; END LAYER 35
LIN {X -34.33, Y -49.21, Z 72.0, A 0, B 90, C 0} C_DIS
WAIT SEC 3
LIN {X -34.33, Y -49.21, Z 74.0, A 0, B 90, C 0} C_DIS
$OUT[1] = TRUE
WAIT SEC 0.8
LIN {X -34.33, Y -49.21, Z 74.0, A 0, B 90, C 0} C_DIS
LIN {X -34.33, Y -49.21, Z 74.0, A 0, B 90, C 0} C_DIS
LIN {X -32.91, Y -50.13, Z 74.0, A 0, B 90, C 0} C_DIS
LIN {X -31.1, Y -51.31, Z 74.0, A 0, B 90, C 0} C_DIS
LIN {X -29.63, Y -52.14, Z 74.0, A 0, B 90, C 0} C_DIS
LIN {X -27.75, Y -53.2, Z 74.0, A 0, B 90, C 0} C_DIS
LIN {X -26.23, Y -53.93, Z 74.0, A 0, B 90, C 0} C_DIS
LIN {X -24.29, Y -54.86, Z 74.0, A 0, B 90, C 0} C_DIS
LIN {X -22.72, Y -55.5, Z 74.0, A 0, B 90, C 0} C_DIS
LIN {X -20.72, Y -56.31, Z 74.0, A 0, B 90, C 0} C_DIS
LIN {X -19.12, Y -56.84, Z 74.0, A 0, B 90, C 0} C_DIS
LIN {X -17.07, Y -57.52, Z 74.0, A 0, B 90, C 0} C_DIS
LIN {X -15.43, Y -57.95, Z 74.0, A 0, B 90, C 0} C_DIS
LIN {X -13.35, Y -58.5, Z 74.0, A 0, B 90, C 0} C_DIS
LIN {X -11.69, Y -58.82, Z 74.0, A 0, B 90, C 0} C_DIS
LIN {X -9.58, Y -59.23, Z 74.0, A 0, B 90, C 0} C_DIS
LIN {X -7.9, Y -59.45, Z 74.0, A 0, B 90, C 0} C_DIS
LIN {X -5.76, Y -59.72, Z 74.0, A 0, B 90, C 0} C_DIS
LIN {X -4.07, Y -59.83, Z 74.0, A 0, B 90, C 0} C_DIS
LIN {X -1.92, Y -59.97, Z 74.0, A 0, B 90, C 0} C_DIS
LIN {X -0.23, Y -59.97, Z 74.0, A 0, B 90, C 0} C_DIS
LIN {X 1.92, Y -59.97, Z 74.0, A 0, B 90, C 0} C_DIS
LIN {X 3.61, Y -59.86, Z 74.0, A 0, B 90, C 0} C_DIS
LIN {X 5.76, Y -59.72, Z 74.0, A 0, B 90, C 0} C_DIS
LIN {X 7.44, Y -59.51, Z 74.0, A 0, B 90, C 0} C_DIS
LIN {X 9.58, Y -59.23, Z 74.0, A 0, B 90, C 0} C_DIS
LIN {X 11.24, Y -58.91, Z 74.0, A 0, B 90, C 0} C_DIS
LIN {X 13.35, Y -58.5, Z 74.0, A 0, B 90, C 0} C_DIS
LIN {X 14.99, Y -58.07, Z 74.0, A 0, B 90, C 0} C_DIS
LIN {X 17.07, Y -57.52, Z 74.0, A 0, B 90, C 0} C_DIS
LIN {X 18.68, Y -56.99, Z 74.0, A 0, B 90, C 0} C_DIS
LIN {X 20.72, Y -56.31, Z 74.0, A 0, B 90, C 0} C_DIS
LIN {X 22.29, Y -55.67, Z 74.0, A 0, B 90, C 0} C_DIS
LIN {X 24.29, Y -54.86, Z 74.0, A 0, B 90, C 0} C_DIS
LIN {X 25.81, Y -54.13, Z 74.0, A 0, B 90, C 0} C_DIS
LIN {X 27.75, Y -53.2, Z 74.0, A 0, B 90, C 0} C_DIS
LIN {X 29.23, Y -52.37, Z 74.0, A 0, B 90, C 0} C_DIS
LIN {X 31.1, Y -51.31, Z 74.0, A 0, B 90, C 0} C_DIS
LIN {X 32.52, Y -50.39, Z 74.0, A 0, B 90, C 0} C_DIS
LIN {X 34.33, Y -49.21, Z 74.0, A 0, B 90, C 0} C_DIS
LIN {X 35.68, Y -48.2, Z 74.0, A 0, B 90, C 0} C_DIS
LIN {X 37.41, Y -46.91, Z 74.0, A 0, B 90, C 0} C_DIS
LIN {X 38.7, Y -45.81, Z 74.0, A 0, B 90, C 0} C_DIS
LIN {X 40.34, Y -44.42, Z 74.0, A 0, B 90, C 0} C_DIS
LIN {X 41.55, Y -43.24, Z 74.0, A 0, B 90, C 0} C_DIS
LIN {X 43.1, Y -41.74, Z 74.0, A 0, B 90, C 0} C_DIS
LIN {X 44.24, Y -40.49, Z 74.0, A 0, B 90, C 0} C_DIS
LIN {X 45.69, Y -38.89, Z 74.0, A 0, B 90, C 0} C_DIS
LIN {X 46.74, Y -37.57, Z 74.0, A 0, B 90, C 0} C_DIS
LIN {X 48.08, Y -35.89, Z 74.0, A 0, B 90, C 0} C_DIS
LIN {X 49.05, Y -34.5, Z 74.0, A 0, B 90, C 0} C_DIS
LIN {X 50.29, Y -32.73, Z 74.0, A 0, B 90, C 0} C_DIS
LIN {X 51.16, Y -31.28, Z 74.0, A 0, B 90, C 0} C_DIS
LIN {X 52.28, Y -29.44, Z 74.0, A 0, B 90, C 0} C_DIS
LIN {X 53.06, Y -27.94, Z 74.0, A 0, B 90, C 0} C_DIS
LIN {X 54.06, Y -26.03, Z 74.0, A 0, B 90, C 0} C_DIS
LIN {X 54.74, Y -24.49, Z 74.0, A 0, B 90, C 0} C_DIS
LIN {X 55.62, Y -22.52, Z 74.0, A 0, B 90, C 0} C_DIS
LIN {X 56.2, Y -20.93, Z 74.0, A 0, B 90, C 0} C_DIS
LIN {X 56.94, Y -18.91, Z 74.0, A 0, B 90, C 0} C_DIS
LIN {X 57.42, Y -17.28, Z 74.0, A 0, B 90, C 0} C_DIS
LIN {X 58.04, Y -15.22, Z 74.0, A 0, B 90, C 0} C_DIS
LIN {X 58.41, Y -13.57, Z 74.0, A 0, B 90, C 0} C_DIS
LIN {X 58.89, Y -11.47, Z 74.0, A 0, B 90, C 0} C_DIS
LIN {X 59.16, Y -9.8, Z 74.0, A 0, B 90, C 0} C_DIS
LIN {X 59.51, Y -7.67, Z 74.0, A 0, B 90, C 0} C_DIS
LIN {X 59.67, Y -5.99, Z 74.0, A 0, B 90, C 0} C_DIS
LIN {X 59.88, Y -3.84, Z 74.0, A 0, B 90, C 0} C_DIS
LIN {X 59.93, Y -2.15, Z 74.0, A 0, B 90, C 0} C_DIS
LIN {X 60.0, Y 0.0, Z 74.0, A 0, B 90, C 0} C_DIS
LIN {X 59.95, Y 1.69, Z 74.0, A 0, B 90, C 0} C_DIS
LIN {X 59.88, Y 3.84, Z 74.0, A 0, B 90, C 0} C_DIS
LIN {X 59.71, Y 5.53, Z 74.0, A 0, B 90, C 0} C_DIS
LIN {X 59.51, Y 7.67, Z 74.0, A 0, B 90, C 0} C_DIS
LIN {X 59.24, Y 9.34, Z 74.0, A 0, B 90, C 0} C_DIS
LIN {X 58.89, Y 11.47, Z 74.0, A 0, B 90, C 0} C_DIS
LIN {X 58.52, Y 13.12, Z 74.0, A 0, B 90, C 0} C_DIS
LIN {X 58.04, Y 15.22, Z 74.0, A 0, B 90, C 0} C_DIS
LIN {X 57.56, Y 16.84, Z 74.0, A 0, B 90, C 0} C_DIS
LIN {X 56.94, Y 18.91, Z 74.0, A 0, B 90, C 0} C_DIS
LIN {X 56.36, Y 20.49, Z 74.0, A 0, B 90, C 0} C_DIS
LIN {X 55.62, Y 22.52, Z 74.0, A 0, B 90, C 0} C_DIS
LIN {X 54.93, Y 24.06, Z 74.0, A 0, B 90, C 0} C_DIS
LIN {X 54.06, Y 26.03, Z 74.0, A 0, B 90, C 0} C_DIS
LIN {X 53.28, Y 27.53, Z 74.0, A 0, B 90, C 0} C_DIS
LIN {X 52.28, Y 29.44, Z 74.0, A 0, B 90, C 0} C_DIS
LIN {X 51.4, Y 30.89, Z 74.0, A 0, B 90, C 0} C_DIS
LIN {X 50.29, Y 32.73, Z 74.0, A 0, B 90, C 0} C_DIS
LIN {X 49.32, Y 34.12, Z 74.0, A 0, B 90, C 0} C_DIS
LIN {X 48.08, Y 35.89, Z 74.0, A 0, B 90, C 0} C_DIS
LIN {X 47.03, Y 37.21, Z 74.0, A 0, B 90, C 0} C_DIS
LIN {X 45.69, Y 38.89, Z 74.0, A 0, B 90, C 0} C_DIS
LIN {X 44.55, Y 40.15, Z 74.0, A 0, B 90, C 0} C_DIS
LIN {X 43.1, Y 41.74, Z 74.0, A 0, B 90, C 0} C_DIS
LIN {X 41.89, Y 42.92, Z 74.0, A 0, B 90, C 0} C_DIS
LIN {X 40.34, Y 44.42, Z 74.0, A 0, B 90, C 0} C_DIS
LIN {X 39.05, Y 45.51, Z 74.0, A 0, B 90, C 0} C_DIS
LIN {X 37.41, Y 46.91, Z 74.0, A 0, B 90, C 0} C_DIS
LIN {X 36.05, Y 47.92, Z 74.0, A 0, B 90, C 0} C_DIS
LIN {X 34.33, Y 49.21, Z 74.0, A 0, B 90, C 0} C_DIS
LIN {X 32.91, Y 50.13, Z 74.0, A 0, B 90, C 0} C_DIS
LIN {X 31.1, Y 51.31, Z 74.0, A 0, B 90, C 0} C_DIS
LIN {X 29.63, Y 52.14, Z 74.0, A 0, B 90, C 0} C_DIS
LIN {X 27.75, Y 53.2, Z 74.0, A 0, B 90, C 0} C_DIS
LIN {X 26.23, Y 53.93, Z 74.0, A 0, B 90, C 0} C_DIS
LIN {X 24.29, Y 54.86, Z 74.0, A 0, B 90, C 0} C_DIS
LIN {X 22.72, Y 55.5, Z 74.0, A 0, B 90, C 0} C_DIS
LIN {X 20.72, Y 56.31, Z 74.0, A 0, B 90, C 0} C_DIS
LIN {X 19.12, Y 56.84, Z 74.0, A 0, B 90, C 0} C_DIS
LIN {X 17.07, Y 57.52, Z 74.0, A 0, B 90, C 0} C_DIS
LIN {X 15.43, Y 57.95, Z 74.0, A 0, B 90, C 0} C_DIS
LIN {X 13.35, Y 58.5, Z 74.0, A 0, B 90, C 0} C_DIS
LIN {X 11.69, Y 58.82, Z 74.0, A 0, B 90, C 0} C_DIS
LIN {X 9.58, Y 59.23, Z 74.0, A 0, B 90, C 0} C_DIS
LIN {X 7.9, Y 59.45, Z 74.0, A 0, B 90, C 0} C_DIS
LIN {X 5.76, Y 59.72, Z 74.0, A 0, B 90, C 0} C_DIS
LIN {X 4.07, Y 59.83, Z 74.0, A 0, B 90, C 0} C_DIS
LIN {X 1.92, Y 59.97, Z 74.0, A 0, B 90, C 0} C_DIS
LIN {X 0.23, Y 59.97, Z 74.0, A 0, B 90, C 0} C_DIS
LIN {X -1.92, Y 59.97, Z 74.0, A 0, B 90, C 0} C_DIS
LIN {X -3.61, Y 59.86, Z 74.0, A 0, B 90, C 0} C_DIS
LIN {X -5.76, Y 59.72, Z 74.0, A 0, B 90, C 0} C_DIS
LIN {X -7.44, Y 59.51, Z 74.0, A 0, B 90, C 0} C_DIS
LIN {X -9.58, Y 59.23, Z 74.0, A 0, B 90, C 0} C_DIS
LIN {X -11.24, Y 58.91, Z 74.0, A 0, B 90, C 0} C_DIS
LIN {X -13.35, Y 58.5, Z 74.0, A 0, B 90, C 0} C_DIS
LIN {X -14.99, Y 58.07, Z 74.0, A 0, B 90, C 0} C_DIS
LIN {X -17.07, Y 57.52, Z 74.0, A 0, B 90, C 0} C_DIS
LIN {X -18.68, Y 56.99, Z 74.0, A 0, B 90, C 0} C_DIS
LIN {X -20.72, Y 56.31, Z 74.0, A 0, B 90, C 0} C_DIS
LIN {X -22.29, Y 55.67, Z 74.0, A 0, B 90, C 0} C_DIS
LIN {X -24.29, Y 54.86, Z 74.0, A 0, B 90, C 0} C_DIS
LIN {X -25.81, Y 54.13, Z 74.0, A 0, B 90, C 0} C_DIS
LIN {X -27.75, Y 53.2, Z 74.0, A 0, B 90, C 0} C_DIS
LIN {X -29.23, Y 52.37, Z 74.0, A 0, B 90, C 0} C_DIS
LIN {X -31.1, Y 51.31, Z 74.0, A 0, B 90, C 0} C_DIS
LIN {X -32.52, Y 50.39, Z 74.0, A 0, B 90, C 0} C_DIS
LIN {X -34.33, Y 49.21, Z 74.0, A 0, B 90, C 0} C_DIS
LIN {X -35.68, Y 48.2, Z 74.0, A 0, B 90, C 0} C_DIS
LIN {X -37.41, Y 46.91, Z 74.0, A 0, B 90, C 0} C_DIS
LIN {X -38.7, Y 45.81, Z 74.0, A 0, B 90, C 0} C_DIS
LIN {X -40.34, Y 44.42, Z 74.0, A 0, B 90, C 0} C_DIS
LIN {X -41.55, Y 43.24, Z 74.0, A 0, B 90, C 0} C_DIS
LIN {X -43.1, Y 41.74, Z 74.0, A 0, B 90, C 0} C_DIS
LIN {X -44.24, Y 40.49, Z 74.0, A 0, B 90, C 0} C_DIS
LIN {X -45.69, Y 38.89, Z 74.0, A 0, B 90, C 0} C_DIS
LIN {X -46.74, Y 37.57, Z 74.0, A 0, B 90, C 0} C_DIS
LIN {X -48.08, Y 35.89, Z 74.0, A 0, B 90, C 0} C_DIS
LIN {X -49.05, Y 34.5, Z 74.0, A 0, B 90, C 0} C_DIS
LIN {X -50.29, Y 32.73, Z 74.0, A 0, B 90, C 0} C_DIS
LIN {X -51.16, Y 31.28, Z 74.0, A 0, B 90, C 0} C_DIS
LIN {X -52.28, Y 29.44, Z 74.0, A 0, B 90, C 0} C_DIS
LIN {X -53.06, Y 27.94, Z 74.0, A 0, B 90, C 0} C_DIS
LIN {X -54.06, Y 26.03, Z 74.0, A 0, B 90, C 0} C_DIS
LIN {X -54.74, Y 24.49, Z 74.0, A 0, B 90, C 0} C_DIS
LIN {X -55.62, Y 22.52, Z 74.0, A 0, B 90, C 0} C_DIS
LIN {X -56.2, Y 20.93, Z 74.0, A 0, B 90, C 0} C_DIS
LIN {X -56.94, Y 18.91, Z 74.0, A 0, B 90, C 0} C_DIS
LIN {X -57.42, Y 17.28, Z 74.0, A 0, B 90, C 0} C_DIS
LIN {X -58.04, Y 15.22, Z 74.0, A 0, B 90, C 0} C_DIS
LIN {X -58.41, Y 13.57, Z 74.0, A 0, B 90, C 0} C_DIS
LIN {X -58.89, Y 11.47, Z 74.0, A 0, B 90, C 0} C_DIS
LIN {X -59.16, Y 9.8, Z 74.0, A 0, B 90, C 0} C_DIS
LIN {X -59.51, Y 7.67, Z 74.0, A 0, B 90, C 0} C_DIS
LIN {X -59.67, Y 5.99, Z 74.0, A 0, B 90, C 0} C_DIS
LIN {X -59.88, Y 3.84, Z 74.0, A 0, B 90, C 0} C_DIS
LIN {X -59.93, Y 2.15, Z 74.0, A 0, B 90, C 0} C_DIS
LIN {X -60.0, Y -0.0, Z 74.0, A 0, B 90, C 0} C_DIS
LIN {X -59.95, Y -1.69, Z 74.0, A 0, B 90, C 0} C_DIS
LIN {X -59.88, Y -3.84, Z 74.0, A 0, B 90, C 0} C_DIS
LIN {X -59.71, Y -5.53, Z 74.0, A 0, B 90, C 0} C_DIS
LIN {X -59.51, Y -7.67, Z 74.0, A 0, B 90, C 0} C_DIS
LIN {X -59.24, Y -9.34, Z 74.0, A 0, B 90, C 0} C_DIS
LIN {X -58.89, Y -11.47, Z 74.0, A 0, B 90, C 0} C_DIS
LIN {X -58.52, Y -13.12, Z 74.0, A 0, B 90, C 0} C_DIS
LIN {X -58.04, Y -15.22, Z 74.0, A 0, B 90, C 0} C_DIS
LIN {X -57.56, Y -16.84, Z 74.0, A 0, B 90, C 0} C_DIS
LIN {X -56.94, Y -18.91, Z 74.0, A 0, B 90, C 0} C_DIS
LIN {X -56.36, Y -20.49, Z 74.0, A 0, B 90, C 0} C_DIS
LIN {X -55.62, Y -22.52, Z 74.0, A 0, B 90, C 0} C_DIS
LIN {X -54.93, Y -24.06, Z 74.0, A 0, B 90, C 0} C_DIS
LIN {X -54.06, Y -26.03, Z 74.0, A 0, B 90, C 0} C_DIS
LIN {X -53.28, Y -27.53, Z 74.0, A 0, B 90, C 0} C_DIS
LIN {X -52.28, Y -29.44, Z 74.0, A 0, B 90, C 0} C_DIS
LIN {X -51.4, Y -30.89, Z 74.0, A 0, B 90, C 0} C_DIS
LIN {X -50.29, Y -32.73, Z 74.0, A 0, B 90, C 0} C_DIS
LIN {X -49.32, Y -34.12, Z 74.0, A 0, B 90, C 0} C_DIS
LIN {X -48.08, Y -35.89, Z 74.0, A 0, B 90, C 0} C_DIS
LIN {X -47.03, Y -37.21, Z 74.0, A 0, B 90, C 0} C_DIS
LIN {X -45.69, Y -38.89, Z 74.0, A 0, B 90, C 0} C_DIS
LIN {X -44.55, Y -40.15, Z 74.0, A 0, B 90, C 0} C_DIS
LIN {X -43.1, Y -41.74, Z 74.0, A 0, B 90, C 0} C_DIS
LIN {X -41.89, Y -42.92, Z 74.0, A 0, B 90, C 0} C_DIS
LIN {X -40.34, Y -44.42, Z 74.0, A 0, B 90, C 0} C_DIS
LIN {X -39.05, Y -45.51, Z 74.0, A 0, B 90, C 0} C_DIS
LIN {X -37.41, Y -46.91, Z 74.0, A 0, B 90, C 0} C_DIS
LIN {X -36.05, Y -47.92, Z 74.0, A 0, B 90, C 0} C_DIS
$OUT[1] = FALSE

; END LAYER 36
LIN {X -34.33, Y -49.21, Z 74.0, A 0, B 90, C 0} C_DIS
WAIT SEC 3
LIN {X -34.33, Y -49.21, Z 76.0, A 0, B 90, C 0} C_DIS
$OUT[1] = TRUE
WAIT SEC 0.8
LIN {X -34.33, Y -49.21, Z 76.0, A 0, B 90, C 0} C_DIS
LIN {X -34.33, Y -49.21, Z 76.0, A 0, B 90, C 0} C_DIS
LIN {X -32.78, Y -50.22, Z 76.0, A 0, B 90, C 0} C_DIS
LIN {X -31.1, Y -51.31, Z 76.0, A 0, B 90, C 0} C_DIS
LIN {X -29.49, Y -52.21, Z 76.0, A 0, B 90, C 0} C_DIS
LIN {X -27.75, Y -53.2, Z 76.0, A 0, B 90, C 0} C_DIS
LIN {X -26.09, Y -54.0, Z 76.0, A 0, B 90, C 0} C_DIS
LIN {X -24.29, Y -54.86, Z 76.0, A 0, B 90, C 0} C_DIS
LIN {X -22.58, Y -55.56, Z 76.0, A 0, B 90, C 0} C_DIS
LIN {X -20.72, Y -56.31, Z 76.0, A 0, B 90, C 0} C_DIS
LIN {X -18.97, Y -56.89, Z 76.0, A 0, B 90, C 0} C_DIS
LIN {X -17.07, Y -57.52, Z 76.0, A 0, B 90, C 0} C_DIS
LIN {X -15.29, Y -57.99, Z 76.0, A 0, B 90, C 0} C_DIS
LIN {X -13.35, Y -58.5, Z 76.0, A 0, B 90, C 0} C_DIS
LIN {X -11.54, Y -58.85, Z 76.0, A 0, B 90, C 0} C_DIS
LIN {X -9.58, Y -59.23, Z 76.0, A 0, B 90, C 0} C_DIS
LIN {X -7.74, Y -59.47, Z 76.0, A 0, B 90, C 0} C_DIS
LIN {X -5.76, Y -59.72, Z 76.0, A 0, B 90, C 0} C_DIS
LIN {X -3.92, Y -59.84, Z 76.0, A 0, B 90, C 0} C_DIS
LIN {X -1.92, Y -59.97, Z 76.0, A 0, B 90, C 0} C_DIS
LIN {X -0.08, Y -59.97, Z 76.0, A 0, B 90, C 0} C_DIS
LIN {X 1.92, Y -59.97, Z 76.0, A 0, B 90, C 0} C_DIS
LIN {X 3.77, Y -59.85, Z 76.0, A 0, B 90, C 0} C_DIS
LIN {X 5.76, Y -59.72, Z 76.0, A 0, B 90, C 0} C_DIS
LIN {X 7.59, Y -59.49, Z 76.0, A 0, B 90, C 0} C_DIS
LIN {X 9.58, Y -59.23, Z 76.0, A 0, B 90, C 0} C_DIS
LIN {X 11.39, Y -58.88, Z 76.0, A 0, B 90, C 0} C_DIS
LIN {X 13.35, Y -58.5, Z 76.0, A 0, B 90, C 0} C_DIS
LIN {X 15.14, Y -58.03, Z 76.0, A 0, B 90, C 0} C_DIS
LIN {X 17.07, Y -57.52, Z 76.0, A 0, B 90, C 0} C_DIS
LIN {X 18.82, Y -56.94, Z 76.0, A 0, B 90, C 0} C_DIS
LIN {X 20.72, Y -56.31, Z 76.0, A 0, B 90, C 0} C_DIS
LIN {X 22.43, Y -55.62, Z 76.0, A 0, B 90, C 0} C_DIS
LIN {X 24.29, Y -54.86, Z 76.0, A 0, B 90, C 0} C_DIS
LIN {X 25.95, Y -54.06, Z 76.0, A 0, B 90, C 0} C_DIS
LIN {X 27.75, Y -53.2, Z 76.0, A 0, B 90, C 0} C_DIS
LIN {X 29.36, Y -52.29, Z 76.0, A 0, B 90, C 0} C_DIS
LIN {X 31.1, Y -51.31, Z 76.0, A 0, B 90, C 0} C_DIS
LIN {X 32.65, Y -50.3, Z 76.0, A 0, B 90, C 0} C_DIS
LIN {X 34.33, Y -49.21, Z 76.0, A 0, B 90, C 0} C_DIS
LIN {X 35.81, Y -48.11, Z 76.0, A 0, B 90, C 0} C_DIS
LIN {X 37.41, Y -46.91, Z 76.0, A 0, B 90, C 0} C_DIS
LIN {X 38.82, Y -45.71, Z 76.0, A 0, B 90, C 0} C_DIS
LIN {X 40.34, Y -44.42, Z 76.0, A 0, B 90, C 0} C_DIS
LIN {X 41.66, Y -43.13, Z 76.0, A 0, B 90, C 0} C_DIS
LIN {X 43.1, Y -41.74, Z 76.0, A 0, B 90, C 0} C_DIS
LIN {X 44.34, Y -40.37, Z 76.0, A 0, B 90, C 0} C_DIS
LIN {X 45.69, Y -38.89, Z 76.0, A 0, B 90, C 0} C_DIS
LIN {X 46.84, Y -37.45, Z 76.0, A 0, B 90, C 0} C_DIS
LIN {X 48.08, Y -35.89, Z 76.0, A 0, B 90, C 0} C_DIS
LIN {X 49.14, Y -34.37, Z 76.0, A 0, B 90, C 0} C_DIS
LIN {X 50.29, Y -32.73, Z 76.0, A 0, B 90, C 0} C_DIS
LIN {X 51.24, Y -31.15, Z 76.0, A 0, B 90, C 0} C_DIS
LIN {X 52.28, Y -29.44, Z 76.0, A 0, B 90, C 0} C_DIS
LIN {X 53.13, Y -27.81, Z 76.0, A 0, B 90, C 0} C_DIS
LIN {X 54.06, Y -26.03, Z 76.0, A 0, B 90, C 0} C_DIS
LIN {X 54.81, Y -24.34, Z 76.0, A 0, B 90, C 0} C_DIS
LIN {X 55.62, Y -22.52, Z 76.0, A 0, B 90, C 0} C_DIS
LIN {X 56.25, Y -20.78, Z 76.0, A 0, B 90, C 0} C_DIS
LIN {X 56.94, Y -18.91, Z 76.0, A 0, B 90, C 0} C_DIS
LIN {X 57.47, Y -17.14, Z 76.0, A 0, B 90, C 0} C_DIS
LIN {X 58.04, Y -15.22, Z 76.0, A 0, B 90, C 0} C_DIS
LIN {X 58.45, Y -13.42, Z 76.0, A 0, B 90, C 0} C_DIS
LIN {X 58.89, Y -11.47, Z 76.0, A 0, B 90, C 0} C_DIS
LIN {X 59.19, Y -9.65, Z 76.0, A 0, B 90, C 0} C_DIS
LIN {X 59.51, Y -7.67, Z 76.0, A 0, B 90, C 0} C_DIS
LIN {X 59.68, Y -5.83, Z 76.0, A 0, B 90, C 0} C_DIS
LIN {X 59.88, Y -3.84, Z 76.0, A 0, B 90, C 0} C_DIS
LIN {X 59.94, Y -2.0, Z 76.0, A 0, B 90, C 0} C_DIS
LIN {X 60.0, Y 0.0, Z 76.0, A 0, B 90, C 0} C_DIS
LIN {X 59.94, Y 1.85, Z 76.0, A 0, B 90, C 0} C_DIS
LIN {X 59.88, Y 3.84, Z 76.0, A 0, B 90, C 0} C_DIS
LIN {X 59.7, Y 5.68, Z 76.0, A 0, B 90, C 0} C_DIS
LIN {X 59.51, Y 7.67, Z 76.0, A 0, B 90, C 0} C_DIS
LIN {X 59.21, Y 9.5, Z 76.0, A 0, B 90, C 0} C_DIS
LIN {X 58.89, Y 11.47, Z 76.0, A 0, B 90, C 0} C_DIS
LIN {X 58.48, Y 13.27, Z 76.0, A 0, B 90, C 0} C_DIS
LIN {X 58.04, Y 15.22, Z 76.0, A 0, B 90, C 0} C_DIS
LIN {X 57.51, Y 16.99, Z 76.0, A 0, B 90, C 0} C_DIS
LIN {X 56.94, Y 18.91, Z 76.0, A 0, B 90, C 0} C_DIS
LIN {X 56.31, Y 20.64, Z 76.0, A 0, B 90, C 0} C_DIS
LIN {X 55.62, Y 22.52, Z 76.0, A 0, B 90, C 0} C_DIS
LIN {X 54.87, Y 24.2, Z 76.0, A 0, B 90, C 0} C_DIS
LIN {X 54.06, Y 26.03, Z 76.0, A 0, B 90, C 0} C_DIS
LIN {X 53.2, Y 27.67, Z 76.0, A 0, B 90, C 0} C_DIS
LIN {X 52.28, Y 29.44, Z 76.0, A 0, B 90, C 0} C_DIS
LIN {X 51.32, Y 31.02, Z 76.0, A 0, B 90, C 0} C_DIS
LIN {X 50.29, Y 32.73, Z 76.0, A 0, B 90, C 0} C_DIS
LIN {X 49.23, Y 34.25, Z 76.0, A 0, B 90, C 0} C_DIS
LIN {X 48.08, Y 35.89, Z 76.0, A 0, B 90, C 0} C_DIS
LIN {X 46.93, Y 37.33, Z 76.0, A 0, B 90, C 0} C_DIS
LIN {X 45.69, Y 38.89, Z 76.0, A 0, B 90, C 0} C_DIS
LIN {X 44.45, Y 40.26, Z 76.0, A 0, B 90, C 0} C_DIS
LIN {X 43.1, Y 41.74, Z 76.0, A 0, B 90, C 0} C_DIS
LIN {X 41.77, Y 43.03, Z 76.0, A 0, B 90, C 0} C_DIS
LIN {X 40.34, Y 44.42, Z 76.0, A 0, B 90, C 0} C_DIS
LIN {X 38.93, Y 45.61, Z 76.0, A 0, B 90, C 0} C_DIS
LIN {X 37.41, Y 46.91, Z 76.0, A 0, B 90, C 0} C_DIS
LIN {X 35.93, Y 48.01, Z 76.0, A 0, B 90, C 0} C_DIS
LIN {X 34.33, Y 49.21, Z 76.0, A 0, B 90, C 0} C_DIS
LIN {X 32.78, Y 50.22, Z 76.0, A 0, B 90, C 0} C_DIS
LIN {X 31.1, Y 51.31, Z 76.0, A 0, B 90, C 0} C_DIS
LIN {X 29.49, Y 52.21, Z 76.0, A 0, B 90, C 0} C_DIS
LIN {X 27.75, Y 53.2, Z 76.0, A 0, B 90, C 0} C_DIS
LIN {X 26.09, Y 54.0, Z 76.0, A 0, B 90, C 0} C_DIS
LIN {X 24.29, Y 54.86, Z 76.0, A 0, B 90, C 0} C_DIS
LIN {X 22.58, Y 55.56, Z 76.0, A 0, B 90, C 0} C_DIS
LIN {X 20.72, Y 56.31, Z 76.0, A 0, B 90, C 0} C_DIS
LIN {X 18.97, Y 56.89, Z 76.0, A 0, B 90, C 0} C_DIS
LIN {X 17.07, Y 57.52, Z 76.0, A 0, B 90, C 0} C_DIS
LIN {X 15.29, Y 57.99, Z 76.0, A 0, B 90, C 0} C_DIS
LIN {X 13.35, Y 58.5, Z 76.0, A 0, B 90, C 0} C_DIS
LIN {X 11.54, Y 58.85, Z 76.0, A 0, B 90, C 0} C_DIS
LIN {X 9.58, Y 59.23, Z 76.0, A 0, B 90, C 0} C_DIS
LIN {X 7.74, Y 59.47, Z 76.0, A 0, B 90, C 0} C_DIS
LIN {X 5.76, Y 59.72, Z 76.0, A 0, B 90, C 0} C_DIS
LIN {X 3.92, Y 59.84, Z 76.0, A 0, B 90, C 0} C_DIS
LIN {X 1.92, Y 59.97, Z 76.0, A 0, B 90, C 0} C_DIS
LIN {X 0.08, Y 59.97, Z 76.0, A 0, B 90, C 0} C_DIS
LIN {X -1.92, Y 59.97, Z 76.0, A 0, B 90, C 0} C_DIS
LIN {X -3.77, Y 59.85, Z 76.0, A 0, B 90, C 0} C_DIS
LIN {X -5.76, Y 59.72, Z 76.0, A 0, B 90, C 0} C_DIS
LIN {X -7.59, Y 59.49, Z 76.0, A 0, B 90, C 0} C_DIS
LIN {X -9.58, Y 59.23, Z 76.0, A 0, B 90, C 0} C_DIS
LIN {X -11.39, Y 58.88, Z 76.0, A 0, B 90, C 0} C_DIS
LIN {X -13.35, Y 58.5, Z 76.0, A 0, B 90, C 0} C_DIS
LIN {X -15.14, Y 58.03, Z 76.0, A 0, B 90, C 0} C_DIS
LIN {X -17.07, Y 57.52, Z 76.0, A 0, B 90, C 0} C_DIS
LIN {X -18.82, Y 56.94, Z 76.0, A 0, B 90, C 0} C_DIS
LIN {X -20.72, Y 56.31, Z 76.0, A 0, B 90, C 0} C_DIS
LIN {X -22.43, Y 55.62, Z 76.0, A 0, B 90, C 0} C_DIS
LIN {X -24.29, Y 54.86, Z 76.0, A 0, B 90, C 0} C_DIS
LIN {X -25.95, Y 54.06, Z 76.0, A 0, B 90, C 0} C_DIS
LIN {X -27.75, Y 53.2, Z 76.0, A 0, B 90, C 0} C_DIS
LIN {X -29.36, Y 52.29, Z 76.0, A 0, B 90, C 0} C_DIS
LIN {X -31.1, Y 51.31, Z 76.0, A 0, B 90, C 0} C_DIS
LIN {X -32.65, Y 50.3, Z 76.0, A 0, B 90, C 0} C_DIS
LIN {X -34.33, Y 49.21, Z 76.0, A 0, B 90, C 0} C_DIS
LIN {X -35.81, Y 48.11, Z 76.0, A 0, B 90, C 0} C_DIS
LIN {X -37.41, Y 46.91, Z 76.0, A 0, B 90, C 0} C_DIS
LIN {X -38.82, Y 45.71, Z 76.0, A 0, B 90, C 0} C_DIS
LIN {X -40.34, Y 44.42, Z 76.0, A 0, B 90, C 0} C_DIS
LIN {X -41.66, Y 43.13, Z 76.0, A 0, B 90, C 0} C_DIS
LIN {X -43.1, Y 41.74, Z 76.0, A 0, B 90, C 0} C_DIS
LIN {X -44.34, Y 40.37, Z 76.0, A 0, B 90, C 0} C_DIS
LIN {X -45.69, Y 38.89, Z 76.0, A 0, B 90, C 0} C_DIS
LIN {X -46.84, Y 37.45, Z 76.0, A 0, B 90, C 0} C_DIS
LIN {X -48.08, Y 35.89, Z 76.0, A 0, B 90, C 0} C_DIS
LIN {X -49.14, Y 34.37, Z 76.0, A 0, B 90, C 0} C_DIS
LIN {X -50.29, Y 32.73, Z 76.0, A 0, B 90, C 0} C_DIS
LIN {X -51.24, Y 31.15, Z 76.0, A 0, B 90, C 0} C_DIS
LIN {X -52.28, Y 29.44, Z 76.0, A 0, B 90, C 0} C_DIS
LIN {X -53.13, Y 27.81, Z 76.0, A 0, B 90, C 0} C_DIS
LIN {X -54.06, Y 26.03, Z 76.0, A 0, B 90, C 0} C_DIS
LIN {X -54.81, Y 24.34, Z 76.0, A 0, B 90, C 0} C_DIS
LIN {X -55.62, Y 22.52, Z 76.0, A 0, B 90, C 0} C_DIS
LIN {X -56.25, Y 20.78, Z 76.0, A 0, B 90, C 0} C_DIS
LIN {X -56.94, Y 18.91, Z 76.0, A 0, B 90, C 0} C_DIS
LIN {X -57.47, Y 17.14, Z 76.0, A 0, B 90, C 0} C_DIS
LIN {X -58.04, Y 15.22, Z 76.0, A 0, B 90, C 0} C_DIS
LIN {X -58.45, Y 13.42, Z 76.0, A 0, B 90, C 0} C_DIS
LIN {X -58.89, Y 11.47, Z 76.0, A 0, B 90, C 0} C_DIS
LIN {X -59.19, Y 9.65, Z 76.0, A 0, B 90, C 0} C_DIS
LIN {X -59.51, Y 7.67, Z 76.0, A 0, B 90, C 0} C_DIS
LIN {X -59.68, Y 5.83, Z 76.0, A 0, B 90, C 0} C_DIS
LIN {X -59.88, Y 3.84, Z 76.0, A 0, B 90, C 0} C_DIS
LIN {X -59.94, Y 2.0, Z 76.0, A 0, B 90, C 0} C_DIS
LIN {X -60.0, Y -0.0, Z 76.0, A 0, B 90, C 0} C_DIS
LIN {X -59.94, Y -1.85, Z 76.0, A 0, B 90, C 0} C_DIS
LIN {X -59.88, Y -3.84, Z 76.0, A 0, B 90, C 0} C_DIS
LIN {X -59.7, Y -5.68, Z 76.0, A 0, B 90, C 0} C_DIS
LIN {X -59.51, Y -7.67, Z 76.0, A 0, B 90, C 0} C_DIS
LIN {X -59.21, Y -9.5, Z 76.0, A 0, B 90, C 0} C_DIS
LIN {X -58.89, Y -11.47, Z 76.0, A 0, B 90, C 0} C_DIS
LIN {X -58.48, Y -13.27, Z 76.0, A 0, B 90, C 0} C_DIS
LIN {X -58.04, Y -15.22, Z 76.0, A 0, B 90, C 0} C_DIS
LIN {X -57.51, Y -16.99, Z 76.0, A 0, B 90, C 0} C_DIS
LIN {X -56.94, Y -18.91, Z 76.0, A 0, B 90, C 0} C_DIS
LIN {X -56.31, Y -20.64, Z 76.0, A 0, B 90, C 0} C_DIS
LIN {X -55.62, Y -22.52, Z 76.0, A 0, B 90, C 0} C_DIS
LIN {X -54.87, Y -24.2, Z 76.0, A 0, B 90, C 0} C_DIS
LIN {X -54.06, Y -26.03, Z 76.0, A 0, B 90, C 0} C_DIS
LIN {X -53.2, Y -27.67, Z 76.0, A 0, B 90, C 0} C_DIS
LIN {X -52.28, Y -29.44, Z 76.0, A 0, B 90, C 0} C_DIS
LIN {X -51.32, Y -31.02, Z 76.0, A 0, B 90, C 0} C_DIS
LIN {X -50.29, Y -32.73, Z 76.0, A 0, B 90, C 0} C_DIS
LIN {X -49.23, Y -34.25, Z 76.0, A 0, B 90, C 0} C_DIS
LIN {X -48.08, Y -35.89, Z 76.0, A 0, B 90, C 0} C_DIS
LIN {X -46.93, Y -37.33, Z 76.0, A 0, B 90, C 0} C_DIS
LIN {X -45.69, Y -38.89, Z 76.0, A 0, B 90, C 0} C_DIS
LIN {X -44.45, Y -40.26, Z 76.0, A 0, B 90, C 0} C_DIS
LIN {X -43.1, Y -41.74, Z 76.0, A 0, B 90, C 0} C_DIS
LIN {X -41.77, Y -43.03, Z 76.0, A 0, B 90, C 0} C_DIS
LIN {X -40.34, Y -44.42, Z 76.0, A 0, B 90, C 0} C_DIS
LIN {X -38.93, Y -45.61, Z 76.0, A 0, B 90, C 0} C_DIS
LIN {X -37.41, Y -46.91, Z 76.0, A 0, B 90, C 0} C_DIS
LIN {X -35.93, Y -48.01, Z 76.0, A 0, B 90, C 0} C_DIS
$OUT[1] = FALSE

; END LAYER 37
LIN {X -34.33, Y -49.21, Z 76.0, A 0, B 90, C 0} C_DIS
WAIT SEC 3
LIN {X -34.33, Y -49.21, Z 78.0, A 0, B 90, C 0} C_DIS
$OUT[1] = TRUE
WAIT SEC 0.8
LIN {X -34.33, Y -49.21, Z 78.0, A 0, B 90, C 0} C_DIS
LIN {X -34.33, Y -49.21, Z 78.0, A 0, B 90, C 0} C_DIS
LIN {X -32.65, Y -50.3, Z 78.0, A 0, B 90, C 0} C_DIS
LIN {X -31.1, Y -51.31, Z 78.0, A 0, B 90, C 0} C_DIS
LIN {X -29.36, Y -52.29, Z 78.0, A 0, B 90, C 0} C_DIS
LIN {X -27.75, Y -53.2, Z 78.0, A 0, B 90, C 0} C_DIS
LIN {X -25.95, Y -54.06, Z 78.0, A 0, B 90, C 0} C_DIS
LIN {X -24.29, Y -54.86, Z 78.0, A 0, B 90, C 0} C_DIS
LIN {X -22.43, Y -55.62, Z 78.0, A 0, B 90, C 0} C_DIS
LIN {X -20.72, Y -56.31, Z 78.0, A 0, B 90, C 0} C_DIS
LIN {X -18.82, Y -56.94, Z 78.0, A 0, B 90, C 0} C_DIS
LIN {X -17.07, Y -57.52, Z 78.0, A 0, B 90, C 0} C_DIS
LIN {X -15.14, Y -58.03, Z 78.0, A 0, B 90, C 0} C_DIS
LIN {X -13.35, Y -58.5, Z 78.0, A 0, B 90, C 0} C_DIS
LIN {X -11.39, Y -58.88, Z 78.0, A 0, B 90, C 0} C_DIS
LIN {X -9.58, Y -59.23, Z 78.0, A 0, B 90, C 0} C_DIS
LIN {X -7.59, Y -59.49, Z 78.0, A 0, B 90, C 0} C_DIS
LIN {X -5.76, Y -59.72, Z 78.0, A 0, B 90, C 0} C_DIS
LIN {X -3.77, Y -59.85, Z 78.0, A 0, B 90, C 0} C_DIS
LIN {X -1.92, Y -59.97, Z 78.0, A 0, B 90, C 0} C_DIS
LIN {X 0.08, Y -59.97, Z 78.0, A 0, B 90, C 0} C_DIS
LIN {X 1.92, Y -59.97, Z 78.0, A 0, B 90, C 0} C_DIS
LIN {X 3.92, Y -59.84, Z 78.0, A 0, B 90, C 0} C_DIS
LIN {X 5.76, Y -59.72, Z 78.0, A 0, B 90, C 0} C_DIS
LIN {X 7.74, Y -59.47, Z 78.0, A 0, B 90, C 0} C_DIS
LIN {X 9.58, Y -59.23, Z 78.0, A 0, B 90, C 0} C_DIS
LIN {X 11.54, Y -58.85, Z 78.0, A 0, B 90, C 0} C_DIS
LIN {X 13.35, Y -58.5, Z 78.0, A 0, B 90, C 0} C_DIS
LIN {X 15.29, Y -57.99, Z 78.0, A 0, B 90, C 0} C_DIS
LIN {X 17.07, Y -57.52, Z 78.0, A 0, B 90, C 0} C_DIS
LIN {X 18.97, Y -56.89, Z 78.0, A 0, B 90, C 0} C_DIS
LIN {X 20.72, Y -56.31, Z 78.0, A 0, B 90, C 0} C_DIS
LIN {X 22.58, Y -55.56, Z 78.0, A 0, B 90, C 0} C_DIS
LIN {X 24.29, Y -54.86, Z 78.0, A 0, B 90, C 0} C_DIS
LIN {X 26.09, Y -54.0, Z 78.0, A 0, B 90, C 0} C_DIS
LIN {X 27.75, Y -53.2, Z 78.0, A 0, B 90, C 0} C_DIS
LIN {X 29.49, Y -52.21, Z 78.0, A 0, B 90, C 0} C_DIS
LIN {X 31.1, Y -51.31, Z 78.0, A 0, B 90, C 0} C_DIS
LIN {X 32.78, Y -50.22, Z 78.0, A 0, B 90, C 0} C_DIS
LIN {X 34.33, Y -49.21, Z 78.0, A 0, B 90, C 0} C_DIS
LIN {X 35.93, Y -48.01, Z 78.0, A 0, B 90, C 0} C_DIS
LIN {X 37.41, Y -46.91, Z 78.0, A 0, B 90, C 0} C_DIS
LIN {X 38.93, Y -45.61, Z 78.0, A 0, B 90, C 0} C_DIS
LIN {X 40.34, Y -44.42, Z 78.0, A 0, B 90, C 0} C_DIS
LIN {X 41.77, Y -43.03, Z 78.0, A 0, B 90, C 0} C_DIS
LIN {X 43.1, Y -41.74, Z 78.0, A 0, B 90, C 0} C_DIS
LIN {X 44.45, Y -40.26, Z 78.0, A 0, B 90, C 0} C_DIS
LIN {X 45.69, Y -38.89, Z 78.0, A 0, B 90, C 0} C_DIS
LIN {X 46.93, Y -37.33, Z 78.0, A 0, B 90, C 0} C_DIS
LIN {X 48.08, Y -35.89, Z 78.0, A 0, B 90, C 0} C_DIS
LIN {X 49.23, Y -34.25, Z 78.0, A 0, B 90, C 0} C_DIS
LIN {X 50.29, Y -32.73, Z 78.0, A 0, B 90, C 0} C_DIS
LIN {X 51.32, Y -31.02, Z 78.0, A 0, B 90, C 0} C_DIS
LIN {X 52.28, Y -29.44, Z 78.0, A 0, B 90, C 0} C_DIS
LIN {X 53.2, Y -27.67, Z 78.0, A 0, B 90, C 0} C_DIS
LIN {X 54.06, Y -26.03, Z 78.0, A 0, B 90, C 0} C_DIS
LIN {X 54.87, Y -24.2, Z 78.0, A 0, B 90, C 0} C_DIS
LIN {X 55.62, Y -22.52, Z 78.0, A 0, B 90, C 0} C_DIS
LIN {X 56.31, Y -20.64, Z 78.0, A 0, B 90, C 0} C_DIS
LIN {X 56.94, Y -18.91, Z 78.0, A 0, B 90, C 0} C_DIS
LIN {X 57.51, Y -16.99, Z 78.0, A 0, B 90, C 0} C_DIS
LIN {X 58.04, Y -15.22, Z 78.0, A 0, B 90, C 0} C_DIS
LIN {X 58.48, Y -13.27, Z 78.0, A 0, B 90, C 0} C_DIS
LIN {X 58.89, Y -11.47, Z 78.0, A 0, B 90, C 0} C_DIS
LIN {X 59.21, Y -9.5, Z 78.0, A 0, B 90, C 0} C_DIS
LIN {X 59.51, Y -7.67, Z 78.0, A 0, B 90, C 0} C_DIS
LIN {X 59.7, Y -5.68, Z 78.0, A 0, B 90, C 0} C_DIS
LIN {X 59.88, Y -3.84, Z 78.0, A 0, B 90, C 0} C_DIS
LIN {X 59.94, Y -1.85, Z 78.0, A 0, B 90, C 0} C_DIS
LIN {X 60.0, Y 0.0, Z 78.0, A 0, B 90, C 0} C_DIS
LIN {X 59.94, Y 2.0, Z 78.0, A 0, B 90, C 0} C_DIS
LIN {X 59.88, Y 3.84, Z 78.0, A 0, B 90, C 0} C_DIS
LIN {X 59.68, Y 5.83, Z 78.0, A 0, B 90, C 0} C_DIS
LIN {X 59.51, Y 7.67, Z 78.0, A 0, B 90, C 0} C_DIS
LIN {X 59.19, Y 9.65, Z 78.0, A 0, B 90, C 0} C_DIS
LIN {X 58.89, Y 11.47, Z 78.0, A 0, B 90, C 0} C_DIS
LIN {X 58.45, Y 13.42, Z 78.0, A 0, B 90, C 0} C_DIS
LIN {X 58.04, Y 15.22, Z 78.0, A 0, B 90, C 0} C_DIS
LIN {X 57.47, Y 17.14, Z 78.0, A 0, B 90, C 0} C_DIS
LIN {X 56.94, Y 18.91, Z 78.0, A 0, B 90, C 0} C_DIS
LIN {X 56.25, Y 20.78, Z 78.0, A 0, B 90, C 0} C_DIS
LIN {X 55.62, Y 22.52, Z 78.0, A 0, B 90, C 0} C_DIS
LIN {X 54.81, Y 24.34, Z 78.0, A 0, B 90, C 0} C_DIS
LIN {X 54.06, Y 26.03, Z 78.0, A 0, B 90, C 0} C_DIS
LIN {X 53.13, Y 27.81, Z 78.0, A 0, B 90, C 0} C_DIS
LIN {X 52.28, Y 29.44, Z 78.0, A 0, B 90, C 0} C_DIS
LIN {X 51.24, Y 31.15, Z 78.0, A 0, B 90, C 0} C_DIS
LIN {X 50.29, Y 32.73, Z 78.0, A 0, B 90, C 0} C_DIS
LIN {X 49.14, Y 34.37, Z 78.0, A 0, B 90, C 0} C_DIS
LIN {X 48.08, Y 35.89, Z 78.0, A 0, B 90, C 0} C_DIS
LIN {X 46.84, Y 37.45, Z 78.0, A 0, B 90, C 0} C_DIS
LIN {X 45.69, Y 38.89, Z 78.0, A 0, B 90, C 0} C_DIS
LIN {X 44.34, Y 40.37, Z 78.0, A 0, B 90, C 0} C_DIS
LIN {X 43.1, Y 41.74, Z 78.0, A 0, B 90, C 0} C_DIS
LIN {X 41.66, Y 43.13, Z 78.0, A 0, B 90, C 0} C_DIS
LIN {X 40.34, Y 44.42, Z 78.0, A 0, B 90, C 0} C_DIS
LIN {X 38.82, Y 45.71, Z 78.0, A 0, B 90, C 0} C_DIS
LIN {X 37.41, Y 46.91, Z 78.0, A 0, B 90, C 0} C_DIS
LIN {X 35.81, Y 48.11, Z 78.0, A 0, B 90, C 0} C_DIS
LIN {X 34.33, Y 49.21, Z 78.0, A 0, B 90, C 0} C_DIS
LIN {X 32.65, Y 50.3, Z 78.0, A 0, B 90, C 0} C_DIS
LIN {X 31.1, Y 51.31, Z 78.0, A 0, B 90, C 0} C_DIS
LIN {X 29.36, Y 52.29, Z 78.0, A 0, B 90, C 0} C_DIS
LIN {X 27.75, Y 53.2, Z 78.0, A 0, B 90, C 0} C_DIS
LIN {X 25.95, Y 54.06, Z 78.0, A 0, B 90, C 0} C_DIS
LIN {X 24.29, Y 54.86, Z 78.0, A 0, B 90, C 0} C_DIS
LIN {X 22.43, Y 55.62, Z 78.0, A 0, B 90, C 0} C_DIS
LIN {X 20.72, Y 56.31, Z 78.0, A 0, B 90, C 0} C_DIS
LIN {X 18.82, Y 56.94, Z 78.0, A 0, B 90, C 0} C_DIS
LIN {X 17.07, Y 57.52, Z 78.0, A 0, B 90, C 0} C_DIS
LIN {X 15.14, Y 58.03, Z 78.0, A 0, B 90, C 0} C_DIS
LIN {X 13.35, Y 58.5, Z 78.0, A 0, B 90, C 0} C_DIS
LIN {X 11.39, Y 58.88, Z 78.0, A 0, B 90, C 0} C_DIS
LIN {X 9.58, Y 59.23, Z 78.0, A 0, B 90, C 0} C_DIS
LIN {X 7.59, Y 59.49, Z 78.0, A 0, B 90, C 0} C_DIS
LIN {X 5.76, Y 59.72, Z 78.0, A 0, B 90, C 0} C_DIS
LIN {X 3.77, Y 59.85, Z 78.0, A 0, B 90, C 0} C_DIS
LIN {X 1.92, Y 59.97, Z 78.0, A 0, B 90, C 0} C_DIS
LIN {X -0.08, Y 59.97, Z 78.0, A 0, B 90, C 0} C_DIS
LIN {X -1.92, Y 59.97, Z 78.0, A 0, B 90, C 0} C_DIS
LIN {X -3.92, Y 59.84, Z 78.0, A 0, B 90, C 0} C_DIS
LIN {X -5.76, Y 59.72, Z 78.0, A 0, B 90, C 0} C_DIS
LIN {X -7.74, Y 59.47, Z 78.0, A 0, B 90, C 0} C_DIS
LIN {X -9.58, Y 59.23, Z 78.0, A 0, B 90, C 0} C_DIS
LIN {X -11.54, Y 58.85, Z 78.0, A 0, B 90, C 0} C_DIS
LIN {X -13.35, Y 58.5, Z 78.0, A 0, B 90, C 0} C_DIS
LIN {X -15.29, Y 57.99, Z 78.0, A 0, B 90, C 0} C_DIS
LIN {X -17.07, Y 57.52, Z 78.0, A 0, B 90, C 0} C_DIS
LIN {X -18.97, Y 56.89, Z 78.0, A 0, B 90, C 0} C_DIS
LIN {X -20.72, Y 56.31, Z 78.0, A 0, B 90, C 0} C_DIS
LIN {X -22.58, Y 55.56, Z 78.0, A 0, B 90, C 0} C_DIS
LIN {X -24.29, Y 54.86, Z 78.0, A 0, B 90, C 0} C_DIS
LIN {X -26.09, Y 54.0, Z 78.0, A 0, B 90, C 0} C_DIS
LIN {X -27.75, Y 53.2, Z 78.0, A 0, B 90, C 0} C_DIS
LIN {X -29.49, Y 52.21, Z 78.0, A 0, B 90, C 0} C_DIS
LIN {X -31.1, Y 51.31, Z 78.0, A 0, B 90, C 0} C_DIS
LIN {X -32.78, Y 50.22, Z 78.0, A 0, B 90, C 0} C_DIS
LIN {X -34.33, Y 49.21, Z 78.0, A 0, B 90, C 0} C_DIS
LIN {X -35.93, Y 48.01, Z 78.0, A 0, B 90, C 0} C_DIS
LIN {X -37.41, Y 46.91, Z 78.0, A 0, B 90, C 0} C_DIS
LIN {X -38.93, Y 45.61, Z 78.0, A 0, B 90, C 0} C_DIS
LIN {X -40.34, Y 44.42, Z 78.0, A 0, B 90, C 0} C_DIS
LIN {X -41.77, Y 43.03, Z 78.0, A 0, B 90, C 0} C_DIS
LIN {X -43.1, Y 41.74, Z 78.0, A 0, B 90, C 0} C_DIS
LIN {X -44.45, Y 40.26, Z 78.0, A 0, B 90, C 0} C_DIS
LIN {X -45.69, Y 38.89, Z 78.0, A 0, B 90, C 0} C_DIS
LIN {X -46.93, Y 37.33, Z 78.0, A 0, B 90, C 0} C_DIS
LIN {X -48.08, Y 35.89, Z 78.0, A 0, B 90, C 0} C_DIS
LIN {X -49.23, Y 34.25, Z 78.0, A 0, B 90, C 0} C_DIS
LIN {X -50.29, Y 32.73, Z 78.0, A 0, B 90, C 0} C_DIS
LIN {X -51.32, Y 31.02, Z 78.0, A 0, B 90, C 0} C_DIS
LIN {X -52.28, Y 29.44, Z 78.0, A 0, B 90, C 0} C_DIS
LIN {X -53.2, Y 27.67, Z 78.0, A 0, B 90, C 0} C_DIS
LIN {X -54.06, Y 26.03, Z 78.0, A 0, B 90, C 0} C_DIS
LIN {X -54.87, Y 24.2, Z 78.0, A 0, B 90, C 0} C_DIS
LIN {X -55.62, Y 22.52, Z 78.0, A 0, B 90, C 0} C_DIS
LIN {X -56.31, Y 20.64, Z 78.0, A 0, B 90, C 0} C_DIS
LIN {X -56.94, Y 18.91, Z 78.0, A 0, B 90, C 0} C_DIS
LIN {X -57.51, Y 16.99, Z 78.0, A 0, B 90, C 0} C_DIS
LIN {X -58.04, Y 15.22, Z 78.0, A 0, B 90, C 0} C_DIS
LIN {X -58.48, Y 13.27, Z 78.0, A 0, B 90, C 0} C_DIS
LIN {X -58.89, Y 11.47, Z 78.0, A 0, B 90, C 0} C_DIS
LIN {X -59.21, Y 9.5, Z 78.0, A 0, B 90, C 0} C_DIS
LIN {X -59.51, Y 7.67, Z 78.0, A 0, B 90, C 0} C_DIS
LIN {X -59.7, Y 5.68, Z 78.0, A 0, B 90, C 0} C_DIS
LIN {X -59.88, Y 3.84, Z 78.0, A 0, B 90, C 0} C_DIS
LIN {X -59.94, Y 1.85, Z 78.0, A 0, B 90, C 0} C_DIS
LIN {X -60.0, Y -0.0, Z 78.0, A 0, B 90, C 0} C_DIS
LIN {X -59.94, Y -2.0, Z 78.0, A 0, B 90, C 0} C_DIS
LIN {X -59.88, Y -3.84, Z 78.0, A 0, B 90, C 0} C_DIS
LIN {X -59.68, Y -5.83, Z 78.0, A 0, B 90, C 0} C_DIS
LIN {X -59.51, Y -7.67, Z 78.0, A 0, B 90, C 0} C_DIS
LIN {X -59.19, Y -9.65, Z 78.0, A 0, B 90, C 0} C_DIS
LIN {X -58.89, Y -11.47, Z 78.0, A 0, B 90, C 0} C_DIS
LIN {X -58.45, Y -13.42, Z 78.0, A 0, B 90, C 0} C_DIS
LIN {X -58.04, Y -15.22, Z 78.0, A 0, B 90, C 0} C_DIS
LIN {X -57.47, Y -17.14, Z 78.0, A 0, B 90, C 0} C_DIS
LIN {X -56.94, Y -18.91, Z 78.0, A 0, B 90, C 0} C_DIS
LIN {X -56.25, Y -20.78, Z 78.0, A 0, B 90, C 0} C_DIS
LIN {X -55.62, Y -22.52, Z 78.0, A 0, B 90, C 0} C_DIS
LIN {X -54.81, Y -24.34, Z 78.0, A 0, B 90, C 0} C_DIS
LIN {X -54.06, Y -26.03, Z 78.0, A 0, B 90, C 0} C_DIS
LIN {X -53.13, Y -27.81, Z 78.0, A 0, B 90, C 0} C_DIS
LIN {X -52.28, Y -29.44, Z 78.0, A 0, B 90, C 0} C_DIS
LIN {X -51.24, Y -31.15, Z 78.0, A 0, B 90, C 0} C_DIS
LIN {X -50.29, Y -32.73, Z 78.0, A 0, B 90, C 0} C_DIS
LIN {X -49.14, Y -34.37, Z 78.0, A 0, B 90, C 0} C_DIS
LIN {X -48.08, Y -35.89, Z 78.0, A 0, B 90, C 0} C_DIS
LIN {X -46.84, Y -37.45, Z 78.0, A 0, B 90, C 0} C_DIS
LIN {X -45.69, Y -38.89, Z 78.0, A 0, B 90, C 0} C_DIS
LIN {X -44.34, Y -40.37, Z 78.0, A 0, B 90, C 0} C_DIS
LIN {X -43.1, Y -41.74, Z 78.0, A 0, B 90, C 0} C_DIS
LIN {X -41.66, Y -43.13, Z 78.0, A 0, B 90, C 0} C_DIS
LIN {X -40.34, Y -44.42, Z 78.0, A 0, B 90, C 0} C_DIS
LIN {X -38.82, Y -45.71, Z 78.0, A 0, B 90, C 0} C_DIS
LIN {X -37.41, Y -46.91, Z 78.0, A 0, B 90, C 0} C_DIS
LIN {X -35.81, Y -48.11, Z 78.0, A 0, B 90, C 0} C_DIS
$OUT[1] = FALSE

; END LAYER 38
LIN {X -34.33, Y -49.21, Z 78.0, A 0, B 90, C 0} C_DIS
WAIT SEC 3
LIN {X -34.33, Y -49.21, Z 80.0, A 0, B 90, C 0} C_DIS
$OUT[1] = TRUE
WAIT SEC 0.8
LIN {X -34.33, Y -49.21, Z 80.0, A 0, B 90, C 0} C_DIS
LIN {X -34.33, Y -49.21, Z 80.0, A 0, B 90, C 0} C_DIS
LIN {X -32.52, Y -50.39, Z 80.0, A 0, B 90, C 0} C_DIS
LIN {X -31.1, Y -51.31, Z 80.0, A 0, B 90, C 0} C_DIS
LIN {X -29.23, Y -52.37, Z 80.0, A 0, B 90, C 0} C_DIS
LIN {X -27.75, Y -53.2, Z 80.0, A 0, B 90, C 0} C_DIS
LIN {X -25.81, Y -54.13, Z 80.0, A 0, B 90, C 0} C_DIS
LIN {X -24.29, Y -54.86, Z 80.0, A 0, B 90, C 0} C_DIS
LIN {X -22.29, Y -55.67, Z 80.0, A 0, B 90, C 0} C_DIS
LIN {X -20.72, Y -56.31, Z 80.0, A 0, B 90, C 0} C_DIS
LIN {X -18.68, Y -56.99, Z 80.0, A 0, B 90, C 0} C_DIS
LIN {X -17.07, Y -57.52, Z 80.0, A 0, B 90, C 0} C_DIS
LIN {X -14.99, Y -58.07, Z 80.0, A 0, B 90, C 0} C_DIS
LIN {X -13.35, Y -58.5, Z 80.0, A 0, B 90, C 0} C_DIS
LIN {X -11.24, Y -58.91, Z 80.0, A 0, B 90, C 0} C_DIS
LIN {X -9.58, Y -59.23, Z 80.0, A 0, B 90, C 0} C_DIS
LIN {X -7.44, Y -59.51, Z 80.0, A 0, B 90, C 0} C_DIS
LIN {X -5.76, Y -59.72, Z 80.0, A 0, B 90, C 0} C_DIS
LIN {X -3.61, Y -59.86, Z 80.0, A 0, B 90, C 0} C_DIS
LIN {X -1.92, Y -59.97, Z 80.0, A 0, B 90, C 0} C_DIS
LIN {X 0.23, Y -59.97, Z 80.0, A 0, B 90, C 0} C_DIS
LIN {X 1.92, Y -59.97, Z 80.0, A 0, B 90, C 0} C_DIS
LIN {X 4.07, Y -59.83, Z 80.0, A 0, B 90, C 0} C_DIS
LIN {X 5.76, Y -59.72, Z 80.0, A 0, B 90, C 0} C_DIS
LIN {X 7.9, Y -59.45, Z 80.0, A 0, B 90, C 0} C_DIS
LIN {X 9.58, Y -59.23, Z 80.0, A 0, B 90, C 0} C_DIS
LIN {X 11.69, Y -58.82, Z 80.0, A 0, B 90, C 0} C_DIS
LIN {X 13.35, Y -58.5, Z 80.0, A 0, B 90, C 0} C_DIS
LIN {X 15.43, Y -57.95, Z 80.0, A 0, B 90, C 0} C_DIS
LIN {X 17.07, Y -57.52, Z 80.0, A 0, B 90, C 0} C_DIS
LIN {X 19.12, Y -56.84, Z 80.0, A 0, B 90, C 0} C_DIS
LIN {X 20.72, Y -56.31, Z 80.0, A 0, B 90, C 0} C_DIS
LIN {X 22.72, Y -55.5, Z 80.0, A 0, B 90, C 0} C_DIS
LIN {X 24.29, Y -54.86, Z 80.0, A 0, B 90, C 0} C_DIS
LIN {X 26.23, Y -53.93, Z 80.0, A 0, B 90, C 0} C_DIS
LIN {X 27.75, Y -53.2, Z 80.0, A 0, B 90, C 0} C_DIS
LIN {X 29.63, Y -52.14, Z 80.0, A 0, B 90, C 0} C_DIS
LIN {X 31.1, Y -51.31, Z 80.0, A 0, B 90, C 0} C_DIS
LIN {X 32.91, Y -50.13, Z 80.0, A 0, B 90, C 0} C_DIS
LIN {X 34.33, Y -49.21, Z 80.0, A 0, B 90, C 0} C_DIS
LIN {X 36.05, Y -47.92, Z 80.0, A 0, B 90, C 0} C_DIS
LIN {X 37.41, Y -46.91, Z 80.0, A 0, B 90, C 0} C_DIS
LIN {X 39.05, Y -45.51, Z 80.0, A 0, B 90, C 0} C_DIS
LIN {X 40.34, Y -44.42, Z 80.0, A 0, B 90, C 0} C_DIS
LIN {X 41.89, Y -42.92, Z 80.0, A 0, B 90, C 0} C_DIS
LIN {X 43.1, Y -41.74, Z 80.0, A 0, B 90, C 0} C_DIS
LIN {X 44.55, Y -40.15, Z 80.0, A 0, B 90, C 0} C_DIS
LIN {X 45.69, Y -38.89, Z 80.0, A 0, B 90, C 0} C_DIS
LIN {X 47.03, Y -37.21, Z 80.0, A 0, B 90, C 0} C_DIS
LIN {X 48.08, Y -35.89, Z 80.0, A 0, B 90, C 0} C_DIS
LIN {X 49.32, Y -34.12, Z 80.0, A 0, B 90, C 0} C_DIS
LIN {X 50.29, Y -32.73, Z 80.0, A 0, B 90, C 0} C_DIS
LIN {X 51.4, Y -30.89, Z 80.0, A 0, B 90, C 0} C_DIS
LIN {X 52.28, Y -29.44, Z 80.0, A 0, B 90, C 0} C_DIS
LIN {X 53.28, Y -27.53, Z 80.0, A 0, B 90, C 0} C_DIS
LIN {X 54.06, Y -26.03, Z 80.0, A 0, B 90, C 0} C_DIS
LIN {X 54.93, Y -24.06, Z 80.0, A 0, B 90, C 0} C_DIS
LIN {X 55.62, Y -22.52, Z 80.0, A 0, B 90, C 0} C_DIS
LIN {X 56.36, Y -20.49, Z 80.0, A 0, B 90, C 0} C_DIS
LIN {X 56.94, Y -18.91, Z 80.0, A 0, B 90, C 0} C_DIS
LIN {X 57.56, Y -16.84, Z 80.0, A 0, B 90, C 0} C_DIS
LIN {X 58.04, Y -15.22, Z 80.0, A 0, B 90, C 0} C_DIS
LIN {X 58.52, Y -13.12, Z 80.0, A 0, B 90, C 0} C_DIS
LIN {X 58.89, Y -11.47, Z 80.0, A 0, B 90, C 0} C_DIS
LIN {X 59.24, Y -9.34, Z 80.0, A 0, B 90, C 0} C_DIS
LIN {X 59.51, Y -7.67, Z 80.0, A 0, B 90, C 0} C_DIS
LIN {X 59.71, Y -5.53, Z 80.0, A 0, B 90, C 0} C_DIS
LIN {X 59.88, Y -3.84, Z 80.0, A 0, B 90, C 0} C_DIS
LIN {X 59.95, Y -1.69, Z 80.0, A 0, B 90, C 0} C_DIS
LIN {X 60.0, Y -0.0, Z 80.0, A 0, B 90, C 0} C_DIS
LIN {X 59.93, Y 2.15, Z 80.0, A 0, B 90, C 0} C_DIS
LIN {X 59.88, Y 3.84, Z 80.0, A 0, B 90, C 0} C_DIS
LIN {X 59.67, Y 5.99, Z 80.0, A 0, B 90, C 0} C_DIS
LIN {X 59.51, Y 7.67, Z 80.0, A 0, B 90, C 0} C_DIS
LIN {X 59.16, Y 9.8, Z 80.0, A 0, B 90, C 0} C_DIS
LIN {X 58.89, Y 11.47, Z 80.0, A 0, B 90, C 0} C_DIS
LIN {X 58.41, Y 13.57, Z 80.0, A 0, B 90, C 0} C_DIS
LIN {X 58.04, Y 15.22, Z 80.0, A 0, B 90, C 0} C_DIS
LIN {X 57.42, Y 17.28, Z 80.0, A 0, B 90, C 0} C_DIS
LIN {X 56.94, Y 18.91, Z 80.0, A 0, B 90, C 0} C_DIS
LIN {X 56.2, Y 20.93, Z 80.0, A 0, B 90, C 0} C_DIS
LIN {X 55.62, Y 22.52, Z 80.0, A 0, B 90, C 0} C_DIS
LIN {X 54.74, Y 24.49, Z 80.0, A 0, B 90, C 0} C_DIS
LIN {X 54.06, Y 26.03, Z 80.0, A 0, B 90, C 0} C_DIS
LIN {X 53.06, Y 27.94, Z 80.0, A 0, B 90, C 0} C_DIS
LIN {X 52.28, Y 29.44, Z 80.0, A 0, B 90, C 0} C_DIS
LIN {X 51.16, Y 31.28, Z 80.0, A 0, B 90, C 0} C_DIS
LIN {X 50.29, Y 32.73, Z 80.0, A 0, B 90, C 0} C_DIS
LIN {X 49.05, Y 34.5, Z 80.0, A 0, B 90, C 0} C_DIS
LIN {X 48.08, Y 35.89, Z 80.0, A 0, B 90, C 0} C_DIS
LIN {X 46.74, Y 37.57, Z 80.0, A 0, B 90, C 0} C_DIS
LIN {X 45.69, Y 38.89, Z 80.0, A 0, B 90, C 0} C_DIS
LIN {X 44.24, Y 40.49, Z 80.0, A 0, B 90, C 0} C_DIS
LIN {X 43.1, Y 41.74, Z 80.0, A 0, B 90, C 0} C_DIS
LIN {X 41.55, Y 43.24, Z 80.0, A 0, B 90, C 0} C_DIS
LIN {X 40.34, Y 44.42, Z 80.0, A 0, B 90, C 0} C_DIS
LIN {X 38.7, Y 45.81, Z 80.0, A 0, B 90, C 0} C_DIS
LIN {X 37.41, Y 46.91, Z 80.0, A 0, B 90, C 0} C_DIS
LIN {X 35.68, Y 48.2, Z 80.0, A 0, B 90, C 0} C_DIS
LIN {X 34.33, Y 49.21, Z 80.0, A 0, B 90, C 0} C_DIS
LIN {X 32.52, Y 50.39, Z 80.0, A 0, B 90, C 0} C_DIS
LIN {X 31.1, Y 51.31, Z 80.0, A 0, B 90, C 0} C_DIS
LIN {X 29.23, Y 52.37, Z 80.0, A 0, B 90, C 0} C_DIS
LIN {X 27.75, Y 53.2, Z 80.0, A 0, B 90, C 0} C_DIS
LIN {X 25.81, Y 54.13, Z 80.0, A 0, B 90, C 0} C_DIS
LIN {X 24.29, Y 54.86, Z 80.0, A 0, B 90, C 0} C_DIS
LIN {X 22.29, Y 55.67, Z 80.0, A 0, B 90, C 0} C_DIS
LIN {X 20.72, Y 56.31, Z 80.0, A 0, B 90, C 0} C_DIS
LIN {X 18.68, Y 56.99, Z 80.0, A 0, B 90, C 0} C_DIS
LIN {X 17.07, Y 57.52, Z 80.0, A 0, B 90, C 0} C_DIS
LIN {X 14.99, Y 58.07, Z 80.0, A 0, B 90, C 0} C_DIS
LIN {X 13.35, Y 58.5, Z 80.0, A 0, B 90, C 0} C_DIS
LIN {X 11.24, Y 58.91, Z 80.0, A 0, B 90, C 0} C_DIS
LIN {X 9.58, Y 59.23, Z 80.0, A 0, B 90, C 0} C_DIS
LIN {X 7.44, Y 59.51, Z 80.0, A 0, B 90, C 0} C_DIS
LIN {X 5.76, Y 59.72, Z 80.0, A 0, B 90, C 0} C_DIS
LIN {X 3.61, Y 59.86, Z 80.0, A 0, B 90, C 0} C_DIS
LIN {X 1.92, Y 59.97, Z 80.0, A 0, B 90, C 0} C_DIS
LIN {X -0.23, Y 59.97, Z 80.0, A 0, B 90, C 0} C_DIS
LIN {X -1.92, Y 59.97, Z 80.0, A 0, B 90, C 0} C_DIS
LIN {X -4.07, Y 59.83, Z 80.0, A 0, B 90, C 0} C_DIS
LIN {X -5.76, Y 59.72, Z 80.0, A 0, B 90, C 0} C_DIS
LIN {X -7.9, Y 59.45, Z 80.0, A 0, B 90, C 0} C_DIS
LIN {X -9.58, Y 59.23, Z 80.0, A 0, B 90, C 0} C_DIS
LIN {X -11.69, Y 58.82, Z 80.0, A 0, B 90, C 0} C_DIS
LIN {X -13.35, Y 58.5, Z 80.0, A 0, B 90, C 0} C_DIS
LIN {X -15.43, Y 57.95, Z 80.0, A 0, B 90, C 0} C_DIS
LIN {X -17.07, Y 57.52, Z 80.0, A 0, B 90, C 0} C_DIS
LIN {X -19.12, Y 56.84, Z 80.0, A 0, B 90, C 0} C_DIS
LIN {X -20.72, Y 56.31, Z 80.0, A 0, B 90, C 0} C_DIS
LIN {X -22.72, Y 55.5, Z 80.0, A 0, B 90, C 0} C_DIS
LIN {X -24.29, Y 54.86, Z 80.0, A 0, B 90, C 0} C_DIS
LIN {X -26.23, Y 53.93, Z 80.0, A 0, B 90, C 0} C_DIS
LIN {X -27.75, Y 53.2, Z 80.0, A 0, B 90, C 0} C_DIS
LIN {X -29.63, Y 52.14, Z 80.0, A 0, B 90, C 0} C_DIS
LIN {X -31.1, Y 51.31, Z 80.0, A 0, B 90, C 0} C_DIS
LIN {X -32.91, Y 50.13, Z 80.0, A 0, B 90, C 0} C_DIS
LIN {X -34.33, Y 49.21, Z 80.0, A 0, B 90, C 0} C_DIS
LIN {X -36.05, Y 47.92, Z 80.0, A 0, B 90, C 0} C_DIS
LIN {X -37.41, Y 46.91, Z 80.0, A 0, B 90, C 0} C_DIS
LIN {X -39.05, Y 45.51, Z 80.0, A 0, B 90, C 0} C_DIS
LIN {X -40.34, Y 44.42, Z 80.0, A 0, B 90, C 0} C_DIS
LIN {X -41.89, Y 42.92, Z 80.0, A 0, B 90, C 0} C_DIS
LIN {X -43.1, Y 41.74, Z 80.0, A 0, B 90, C 0} C_DIS
LIN {X -44.55, Y 40.15, Z 80.0, A 0, B 90, C 0} C_DIS
LIN {X -45.69, Y 38.89, Z 80.0, A 0, B 90, C 0} C_DIS
LIN {X -47.03, Y 37.21, Z 80.0, A 0, B 90, C 0} C_DIS
LIN {X -48.08, Y 35.89, Z 80.0, A 0, B 90, C 0} C_DIS
LIN {X -49.32, Y 34.12, Z 80.0, A 0, B 90, C 0} C_DIS
LIN {X -50.29, Y 32.73, Z 80.0, A 0, B 90, C 0} C_DIS
LIN {X -51.4, Y 30.89, Z 80.0, A 0, B 90, C 0} C_DIS
LIN {X -52.28, Y 29.44, Z 80.0, A 0, B 90, C 0} C_DIS
LIN {X -53.28, Y 27.53, Z 80.0, A 0, B 90, C 0} C_DIS
LIN {X -54.06, Y 26.03, Z 80.0, A 0, B 90, C 0} C_DIS
LIN {X -54.93, Y 24.06, Z 80.0, A 0, B 90, C 0} C_DIS
LIN {X -55.62, Y 22.52, Z 80.0, A 0, B 90, C 0} C_DIS
LIN {X -56.36, Y 20.49, Z 80.0, A 0, B 90, C 0} C_DIS
LIN {X -56.94, Y 18.91, Z 80.0, A 0, B 90, C 0} C_DIS
LIN {X -57.56, Y 16.84, Z 80.0, A 0, B 90, C 0} C_DIS
LIN {X -58.04, Y 15.22, Z 80.0, A 0, B 90, C 0} C_DIS
LIN {X -58.52, Y 13.12, Z 80.0, A 0, B 90, C 0} C_DIS
LIN {X -58.89, Y 11.47, Z 80.0, A 0, B 90, C 0} C_DIS
LIN {X -59.24, Y 9.34, Z 80.0, A 0, B 90, C 0} C_DIS
LIN {X -59.51, Y 7.67, Z 80.0, A 0, B 90, C 0} C_DIS
LIN {X -59.71, Y 5.53, Z 80.0, A 0, B 90, C 0} C_DIS
LIN {X -59.88, Y 3.84, Z 80.0, A 0, B 90, C 0} C_DIS
LIN {X -59.95, Y 1.69, Z 80.0, A 0, B 90, C 0} C_DIS
LIN {X -60.0, Y -0.0, Z 80.0, A 0, B 90, C 0} C_DIS
LIN {X -59.93, Y -2.15, Z 80.0, A 0, B 90, C 0} C_DIS
LIN {X -59.88, Y -3.84, Z 80.0, A 0, B 90, C 0} C_DIS
LIN {X -59.67, Y -5.99, Z 80.0, A 0, B 90, C 0} C_DIS
LIN {X -59.51, Y -7.67, Z 80.0, A 0, B 90, C 0} C_DIS
LIN {X -59.16, Y -9.8, Z 80.0, A 0, B 90, C 0} C_DIS
LIN {X -58.89, Y -11.47, Z 80.0, A 0, B 90, C 0} C_DIS
LIN {X -58.41, Y -13.57, Z 80.0, A 0, B 90, C 0} C_DIS
LIN {X -58.04, Y -15.22, Z 80.0, A 0, B 90, C 0} C_DIS
LIN {X -57.42, Y -17.28, Z 80.0, A 0, B 90, C 0} C_DIS
LIN {X -56.94, Y -18.91, Z 80.0, A 0, B 90, C 0} C_DIS
LIN {X -56.2, Y -20.93, Z 80.0, A 0, B 90, C 0} C_DIS
LIN {X -55.62, Y -22.52, Z 80.0, A 0, B 90, C 0} C_DIS
LIN {X -54.74, Y -24.49, Z 80.0, A 0, B 90, C 0} C_DIS
LIN {X -54.06, Y -26.03, Z 80.0, A 0, B 90, C 0} C_DIS
LIN {X -53.06, Y -27.94, Z 80.0, A 0, B 90, C 0} C_DIS
LIN {X -52.28, Y -29.44, Z 80.0, A 0, B 90, C 0} C_DIS
LIN {X -51.16, Y -31.28, Z 80.0, A 0, B 90, C 0} C_DIS
LIN {X -50.29, Y -32.73, Z 80.0, A 0, B 90, C 0} C_DIS
LIN {X -49.05, Y -34.5, Z 80.0, A 0, B 90, C 0} C_DIS
LIN {X -48.08, Y -35.89, Z 80.0, A 0, B 90, C 0} C_DIS
LIN {X -46.74, Y -37.57, Z 80.0, A 0, B 90, C 0} C_DIS
LIN {X -45.69, Y -38.89, Z 80.0, A 0, B 90, C 0} C_DIS
LIN {X -44.24, Y -40.49, Z 80.0, A 0, B 90, C 0} C_DIS
LIN {X -43.1, Y -41.74, Z 80.0, A 0, B 90, C 0} C_DIS
LIN {X -41.55, Y -43.24, Z 80.0, A 0, B 90, C 0} C_DIS
LIN {X -40.34, Y -44.42, Z 80.0, A 0, B 90, C 0} C_DIS
LIN {X -38.7, Y -45.81, Z 80.0, A 0, B 90, C 0} C_DIS
LIN {X -37.41, Y -46.91, Z 80.0, A 0, B 90, C 0} C_DIS
LIN {X -35.68, Y -48.2, Z 80.0, A 0, B 90, C 0} C_DIS
$OUT[1] = FALSE

; END LAYER 39
LIN {X -34.33, Y -49.21, Z 80.0, A 0, B 90, C 0} C_DIS
WAIT SEC 3
LIN {X -34.33, Y -49.21, Z 82.0, A 0, B 90, C 0} C_DIS
$OUT[1] = TRUE
WAIT SEC 0.8
LIN {X -34.33, Y -49.21, Z 82.0, A 0, B 90, C 0} C_DIS
LIN {X -34.33, Y -49.21, Z 82.0, A 0, B 90, C 0} C_DIS
LIN {X -32.39, Y -50.47, Z 82.0, A 0, B 90, C 0} C_DIS
LIN {X -31.1, Y -51.31, Z 82.0, A 0, B 90, C 0} C_DIS
LIN {X -29.09, Y -52.44, Z 82.0, A 0, B 90, C 0} C_DIS
LIN {X -27.75, Y -53.2, Z 82.0, A 0, B 90, C 0} C_DIS
LIN {X -25.67, Y -54.2, Z 82.0, A 0, B 90, C 0} C_DIS
LIN {X -24.29, Y -54.86, Z 82.0, A 0, B 90, C 0} C_DIS
LIN {X -22.15, Y -55.73, Z 82.0, A 0, B 90, C 0} C_DIS
LIN {X -20.72, Y -56.31, Z 82.0, A 0, B 90, C 0} C_DIS
LIN {X -18.53, Y -57.04, Z 82.0, A 0, B 90, C 0} C_DIS
LIN {X -17.07, Y -57.52, Z 82.0, A 0, B 90, C 0} C_DIS
LIN {X -14.84, Y -58.11, Z 82.0, A 0, B 90, C 0} C_DIS
LIN {X -13.35, Y -58.5, Z 82.0, A 0, B 90, C 0} C_DIS
LIN {X -11.09, Y -58.94, Z 82.0, A 0, B 90, C 0} C_DIS
LIN {X -9.58, Y -59.23, Z 82.0, A 0, B 90, C 0} C_DIS
LIN {X -7.29, Y -59.53, Z 82.0, A 0, B 90, C 0} C_DIS
LIN {X -5.76, Y -59.72, Z 82.0, A 0, B 90, C 0} C_DIS
LIN {X -3.46, Y -59.87, Z 82.0, A 0, B 90, C 0} C_DIS
LIN {X -1.92, Y -59.97, Z 82.0, A 0, B 90, C 0} C_DIS
LIN {X 0.38, Y -59.97, Z 82.0, A 0, B 90, C 0} C_DIS
LIN {X 1.92, Y -59.97, Z 82.0, A 0, B 90, C 0} C_DIS
LIN {X 4.23, Y -59.82, Z 82.0, A 0, B 90, C 0} C_DIS
LIN {X 5.76, Y -59.72, Z 82.0, A 0, B 90, C 0} C_DIS
LIN {X 8.05, Y -59.43, Z 82.0, A 0, B 90, C 0} C_DIS
LIN {X 9.58, Y -59.23, Z 82.0, A 0, B 90, C 0} C_DIS
LIN {X 11.84, Y -58.79, Z 82.0, A 0, B 90, C 0} C_DIS
LIN {X 13.35, Y -58.5, Z 82.0, A 0, B 90, C 0} C_DIS
LIN {X 15.58, Y -57.91, Z 82.0, A 0, B 90, C 0} C_DIS
LIN {X 17.07, Y -57.52, Z 82.0, A 0, B 90, C 0} C_DIS
LIN {X 19.26, Y -56.79, Z 82.0, A 0, B 90, C 0} C_DIS
LIN {X 20.72, Y -56.31, Z 82.0, A 0, B 90, C 0} C_DIS
LIN {X 22.86, Y -55.44, Z 82.0, A 0, B 90, C 0} C_DIS
LIN {X 24.29, Y -54.86, Z 82.0, A 0, B 90, C 0} C_DIS
LIN {X 26.37, Y -53.86, Z 82.0, A 0, B 90, C 0} C_DIS
LIN {X 27.75, Y -53.2, Z 82.0, A 0, B 90, C 0} C_DIS
LIN {X 29.76, Y -52.06, Z 82.0, A 0, B 90, C 0} C_DIS
LIN {X 31.1, Y -51.31, Z 82.0, A 0, B 90, C 0} C_DIS
LIN {X 33.04, Y -50.05, Z 82.0, A 0, B 90, C 0} C_DIS
LIN {X 34.33, Y -49.21, Z 82.0, A 0, B 90, C 0} C_DIS
LIN {X 36.18, Y -47.83, Z 82.0, A 0, B 90, C 0} C_DIS
LIN {X 37.41, Y -46.91, Z 82.0, A 0, B 90, C 0} C_DIS
LIN {X 39.17, Y -45.41, Z 82.0, A 0, B 90, C 0} C_DIS
LIN {X 40.34, Y -44.42, Z 82.0, A 0, B 90, C 0} C_DIS
LIN {X 42.0, Y -42.81, Z 82.0, A 0, B 90, C 0} C_DIS
LIN {X 43.1, Y -41.74, Z 82.0, A 0, B 90, C 0} C_DIS
LIN {X 44.65, Y -40.03, Z 82.0, A 0, B 90, C 0} C_DIS
LIN {X 45.69, Y -38.89, Z 82.0, A 0, B 90, C 0} C_DIS
LIN {X 47.13, Y -37.09, Z 82.0, A 0, B 90, C 0} C_DIS
LIN {X 48.08, Y -35.89, Z 82.0, A 0, B 90, C 0} C_DIS
LIN {X 49.41, Y -33.99, Z 82.0, A 0, B 90, C 0} C_DIS
LIN {X 50.29, Y -32.73, Z 82.0, A 0, B 90, C 0} C_DIS
LIN {X 51.48, Y -30.76, Z 82.0, A 0, B 90, C 0} C_DIS
LIN {X 52.28, Y -29.44, Z 82.0, A 0, B 90, C 0} C_DIS
LIN {X 53.35, Y -27.4, Z 82.0, A 0, B 90, C 0} C_DIS
LIN {X 54.06, Y -26.03, Z 82.0, A 0, B 90, C 0} C_DIS
LIN {X 54.99, Y -23.92, Z 82.0, A 0, B 90, C 0} C_DIS
LIN {X 55.62, Y -22.52, Z 82.0, A 0, B 90, C 0} C_DIS
LIN {X 56.41, Y -20.35, Z 82.0, A 0, B 90, C 0} C_DIS
LIN {X 56.94, Y -18.91, Z 82.0, A 0, B 90, C 0} C_DIS
LIN {X 57.6, Y -16.69, Z 82.0, A 0, B 90, C 0} C_DIS
LIN {X 58.04, Y -15.22, Z 82.0, A 0, B 90, C 0} C_DIS
LIN {X 58.55, Y -12.97, Z 82.0, A 0, B 90, C 0} C_DIS
LIN {X 58.89, Y -11.47, Z 82.0, A 0, B 90, C 0} C_DIS
LIN {X 59.26, Y -9.19, Z 82.0, A 0, B 90, C 0} C_DIS
LIN {X 59.51, Y -7.67, Z 82.0, A 0, B 90, C 0} C_DIS
LIN {X 59.73, Y -5.38, Z 82.0, A 0, B 90, C 0} C_DIS
LIN {X 59.88, Y -3.84, Z 82.0, A 0, B 90, C 0} C_DIS
LIN {X 59.95, Y -1.54, Z 82.0, A 0, B 90, C 0} C_DIS
LIN {X 60.0, Y -0.0, Z 82.0, A 0, B 90, C 0} C_DIS
LIN {X 59.93, Y 2.31, Z 82.0, A 0, B 90, C 0} C_DIS
LIN {X 59.88, Y 3.84, Z 82.0, A 0, B 90, C 0} C_DIS
LIN {X 59.66, Y 6.14, Z 82.0, A 0, B 90, C 0} C_DIS
LIN {X 59.51, Y 7.67, Z 82.0, A 0, B 90, C 0} C_DIS
LIN {X 59.14, Y 9.95, Z 82.0, A 0, B 90, C 0} C_DIS
LIN {X 58.89, Y 11.47, Z 82.0, A 0, B 90, C 0} C_DIS
LIN {X 58.38, Y 13.72, Z 82.0, A 0, B 90, C 0} C_DIS
LIN {X 58.04, Y 15.22, Z 82.0, A 0, B 90, C 0} C_DIS
LIN {X 57.38, Y 17.43, Z 82.0, A 0, B 90, C 0} C_DIS
LIN {X 56.94, Y 18.91, Z 82.0, A 0, B 90, C 0} C_DIS
LIN {X 56.15, Y 21.07, Z 82.0, A 0, B 90, C 0} C_DIS
LIN {X 55.62, Y 22.52, Z 82.0, A 0, B 90, C 0} C_DIS
LIN {X 54.68, Y 24.63, Z 82.0, A 0, B 90, C 0} C_DIS
LIN {X 54.06, Y 26.03, Z 82.0, A 0, B 90, C 0} C_DIS
LIN {X 52.99, Y 28.08, Z 82.0, A 0, B 90, C 0} C_DIS
LIN {X 52.28, Y 29.44, Z 82.0, A 0, B 90, C 0} C_DIS
LIN {X 51.08, Y 31.42, Z 82.0, A 0, B 90, C 0} C_DIS
LIN {X 50.29, Y 32.73, Z 82.0, A 0, B 90, C 0} C_DIS
LIN {X 48.97, Y 34.62, Z 82.0, A 0, B 90, C 0} C_DIS
LIN {X 48.08, Y 35.89, Z 82.0, A 0, B 90, C 0} C_DIS
LIN {X 46.65, Y 37.69, Z 82.0, A 0, B 90, C 0} C_DIS
LIN {X 45.69, Y 38.89, Z 82.0, A 0, B 90, C 0} C_DIS
LIN {X 44.14, Y 40.6, Z 82.0, A 0, B 90, C 0} C_DIS
LIN {X 43.1, Y 41.74, Z 82.0, A 0, B 90, C 0} C_DIS
LIN {X 41.44, Y 43.35, Z 82.0, A 0, B 90, C 0} C_DIS
LIN {X 40.34, Y 44.42, Z 82.0, A 0, B 90, C 0} C_DIS
LIN {X 38.58, Y 45.91, Z 82.0, A 0, B 90, C 0} C_DIS
LIN {X 37.41, Y 46.91, Z 82.0, A 0, B 90, C 0} C_DIS
LIN {X 35.56, Y 48.29, Z 82.0, A 0, B 90, C 0} C_DIS
LIN {X 34.33, Y 49.21, Z 82.0, A 0, B 90, C 0} C_DIS
LIN {X 32.39, Y 50.47, Z 82.0, A 0, B 90, C 0} C_DIS
LIN {X 31.1, Y 51.31, Z 82.0, A 0, B 90, C 0} C_DIS
LIN {X 29.09, Y 52.44, Z 82.0, A 0, B 90, C 0} C_DIS
LIN {X 27.75, Y 53.2, Z 82.0, A 0, B 90, C 0} C_DIS
LIN {X 25.67, Y 54.2, Z 82.0, A 0, B 90, C 0} C_DIS
LIN {X 24.29, Y 54.86, Z 82.0, A 0, B 90, C 0} C_DIS
LIN {X 22.15, Y 55.73, Z 82.0, A 0, B 90, C 0} C_DIS
LIN {X 20.72, Y 56.31, Z 82.0, A 0, B 90, C 0} C_DIS
LIN {X 18.53, Y 57.04, Z 82.0, A 0, B 90, C 0} C_DIS
LIN {X 17.07, Y 57.52, Z 82.0, A 0, B 90, C 0} C_DIS
LIN {X 14.84, Y 58.11, Z 82.0, A 0, B 90, C 0} C_DIS
LIN {X 13.35, Y 58.5, Z 82.0, A 0, B 90, C 0} C_DIS
LIN {X 11.09, Y 58.94, Z 82.0, A 0, B 90, C 0} C_DIS
LIN {X 9.58, Y 59.23, Z 82.0, A 0, B 90, C 0} C_DIS
LIN {X 7.29, Y 59.53, Z 82.0, A 0, B 90, C 0} C_DIS
LIN {X 5.76, Y 59.72, Z 82.0, A 0, B 90, C 0} C_DIS
LIN {X 3.46, Y 59.87, Z 82.0, A 0, B 90, C 0} C_DIS
LIN {X 1.92, Y 59.97, Z 82.0, A 0, B 90, C 0} C_DIS
LIN {X -0.38, Y 59.97, Z 82.0, A 0, B 90, C 0} C_DIS
LIN {X -1.92, Y 59.97, Z 82.0, A 0, B 90, C 0} C_DIS
LIN {X -4.23, Y 59.82, Z 82.0, A 0, B 90, C 0} C_DIS
LIN {X -5.76, Y 59.72, Z 82.0, A 0, B 90, C 0} C_DIS
LIN {X -8.05, Y 59.43, Z 82.0, A 0, B 90, C 0} C_DIS
LIN {X -9.58, Y 59.23, Z 82.0, A 0, B 90, C 0} C_DIS
LIN {X -11.84, Y 58.79, Z 82.0, A 0, B 90, C 0} C_DIS
LIN {X -13.35, Y 58.5, Z 82.0, A 0, B 90, C 0} C_DIS
LIN {X -15.58, Y 57.91, Z 82.0, A 0, B 90, C 0} C_DIS
LIN {X -17.07, Y 57.52, Z 82.0, A 0, B 90, C 0} C_DIS
LIN {X -19.26, Y 56.79, Z 82.0, A 0, B 90, C 0} C_DIS
LIN {X -20.72, Y 56.31, Z 82.0, A 0, B 90, C 0} C_DIS
LIN {X -22.86, Y 55.44, Z 82.0, A 0, B 90, C 0} C_DIS
LIN {X -24.29, Y 54.86, Z 82.0, A 0, B 90, C 0} C_DIS
LIN {X -26.37, Y 53.86, Z 82.0, A 0, B 90, C 0} C_DIS
LIN {X -27.75, Y 53.2, Z 82.0, A 0, B 90, C 0} C_DIS
LIN {X -29.76, Y 52.06, Z 82.0, A 0, B 90, C 0} C_DIS
LIN {X -31.1, Y 51.31, Z 82.0, A 0, B 90, C 0} C_DIS
LIN {X -33.04, Y 50.05, Z 82.0, A 0, B 90, C 0} C_DIS
LIN {X -34.33, Y 49.21, Z 82.0, A 0, B 90, C 0} C_DIS
LIN {X -36.18, Y 47.83, Z 82.0, A 0, B 90, C 0} C_DIS
LIN {X -37.41, Y 46.91, Z 82.0, A 0, B 90, C 0} C_DIS
LIN {X -39.17, Y 45.41, Z 82.0, A 0, B 90, C 0} C_DIS
LIN {X -40.34, Y 44.42, Z 82.0, A 0, B 90, C 0} C_DIS
LIN {X -42.0, Y 42.81, Z 82.0, A 0, B 90, C 0} C_DIS
LIN {X -43.1, Y 41.74, Z 82.0, A 0, B 90, C 0} C_DIS
LIN {X -44.65, Y 40.03, Z 82.0, A 0, B 90, C 0} C_DIS
LIN {X -45.69, Y 38.89, Z 82.0, A 0, B 90, C 0} C_DIS
LIN {X -47.13, Y 37.09, Z 82.0, A 0, B 90, C 0} C_DIS
LIN {X -48.08, Y 35.89, Z 82.0, A 0, B 90, C 0} C_DIS
LIN {X -49.41, Y 33.99, Z 82.0, A 0, B 90, C 0} C_DIS
LIN {X -50.29, Y 32.73, Z 82.0, A 0, B 90, C 0} C_DIS
LIN {X -51.48, Y 30.76, Z 82.0, A 0, B 90, C 0} C_DIS
LIN {X -52.28, Y 29.44, Z 82.0, A 0, B 90, C 0} C_DIS
LIN {X -53.35, Y 27.4, Z 82.0, A 0, B 90, C 0} C_DIS
LIN {X -54.06, Y 26.03, Z 82.0, A 0, B 90, C 0} C_DIS
LIN {X -54.99, Y 23.92, Z 82.0, A 0, B 90, C 0} C_DIS
LIN {X -55.62, Y 22.52, Z 82.0, A 0, B 90, C 0} C_DIS
LIN {X -56.41, Y 20.35, Z 82.0, A 0, B 90, C 0} C_DIS
LIN {X -56.94, Y 18.91, Z 82.0, A 0, B 90, C 0} C_DIS
LIN {X -57.6, Y 16.69, Z 82.0, A 0, B 90, C 0} C_DIS
LIN {X -58.04, Y 15.22, Z 82.0, A 0, B 90, C 0} C_DIS
LIN {X -58.55, Y 12.97, Z 82.0, A 0, B 90, C 0} C_DIS
LIN {X -58.89, Y 11.47, Z 82.0, A 0, B 90, C 0} C_DIS
LIN {X -59.26, Y 9.19, Z 82.0, A 0, B 90, C 0} C_DIS
LIN {X -59.51, Y 7.67, Z 82.0, A 0, B 90, C 0} C_DIS
LIN {X -59.73, Y 5.38, Z 82.0, A 0, B 90, C 0} C_DIS
LIN {X -59.88, Y 3.84, Z 82.0, A 0, B 90, C 0} C_DIS
LIN {X -59.95, Y 1.54, Z 82.0, A 0, B 90, C 0} C_DIS
LIN {X -60.0, Y -0.0, Z 82.0, A 0, B 90, C 0} C_DIS
LIN {X -59.93, Y -2.31, Z 82.0, A 0, B 90, C 0} C_DIS
LIN {X -59.88, Y -3.84, Z 82.0, A 0, B 90, C 0} C_DIS
LIN {X -59.66, Y -6.14, Z 82.0, A 0, B 90, C 0} C_DIS
LIN {X -59.51, Y -7.67, Z 82.0, A 0, B 90, C 0} C_DIS
LIN {X -59.14, Y -9.95, Z 82.0, A 0, B 90, C 0} C_DIS
LIN {X -58.89, Y -11.47, Z 82.0, A 0, B 90, C 0} C_DIS
LIN {X -58.38, Y -13.72, Z 82.0, A 0, B 90, C 0} C_DIS
LIN {X -58.04, Y -15.22, Z 82.0, A 0, B 90, C 0} C_DIS
LIN {X -57.38, Y -17.43, Z 82.0, A 0, B 90, C 0} C_DIS
LIN {X -56.94, Y -18.91, Z 82.0, A 0, B 90, C 0} C_DIS
LIN {X -56.15, Y -21.07, Z 82.0, A 0, B 90, C 0} C_DIS
LIN {X -55.62, Y -22.52, Z 82.0, A 0, B 90, C 0} C_DIS
LIN {X -54.68, Y -24.63, Z 82.0, A 0, B 90, C 0} C_DIS
LIN {X -54.06, Y -26.03, Z 82.0, A 0, B 90, C 0} C_DIS
LIN {X -52.99, Y -28.08, Z 82.0, A 0, B 90, C 0} C_DIS
LIN {X -52.28, Y -29.44, Z 82.0, A 0, B 90, C 0} C_DIS
LIN {X -51.08, Y -31.42, Z 82.0, A 0, B 90, C 0} C_DIS
LIN {X -50.29, Y -32.73, Z 82.0, A 0, B 90, C 0} C_DIS
LIN {X -48.97, Y -34.62, Z 82.0, A 0, B 90, C 0} C_DIS
LIN {X -48.08, Y -35.89, Z 82.0, A 0, B 90, C 0} C_DIS
LIN {X -46.65, Y -37.69, Z 82.0, A 0, B 90, C 0} C_DIS
LIN {X -45.69, Y -38.89, Z 82.0, A 0, B 90, C 0} C_DIS
LIN {X -44.14, Y -40.6, Z 82.0, A 0, B 90, C 0} C_DIS
LIN {X -43.1, Y -41.74, Z 82.0, A 0, B 90, C 0} C_DIS
LIN {X -41.44, Y -43.35, Z 82.0, A 0, B 90, C 0} C_DIS
LIN {X -40.34, Y -44.42, Z 82.0, A 0, B 90, C 0} C_DIS
LIN {X -38.58, Y -45.91, Z 82.0, A 0, B 90, C 0} C_DIS
LIN {X -37.41, Y -46.91, Z 82.0, A 0, B 90, C 0} C_DIS
LIN {X -35.56, Y -48.29, Z 82.0, A 0, B 90, C 0} C_DIS
$OUT[1] = FALSE

; END LAYER 40
LIN {X -34.33, Y -49.21, Z 82.0, A 0, B 90, C 0} C_DIS
WAIT SEC 3
LIN {X -34.33, Y -49.21, Z 84.0, A 0, B 90, C 0} C_DIS
$OUT[1] = TRUE
WAIT SEC 0.8
LIN {X -34.33, Y -49.21, Z 84.0, A 0, B 90, C 0} C_DIS
LIN {X -34.33, Y -49.21, Z 84.0, A 0, B 90, C 0} C_DIS
LIN {X -32.26, Y -50.55, Z 84.0, A 0, B 90, C 0} C_DIS
LIN {X -31.1, Y -51.31, Z 84.0, A 0, B 90, C 0} C_DIS
LIN {X -28.96, Y -52.52, Z 84.0, A 0, B 90, C 0} C_DIS
LIN {X -27.75, Y -53.2, Z 84.0, A 0, B 90, C 0} C_DIS
LIN {X -25.53, Y -54.26, Z 84.0, A 0, B 90, C 0} C_DIS
LIN {X -24.29, Y -54.86, Z 84.0, A 0, B 90, C 0} C_DIS
LIN {X -22.01, Y -55.79, Z 84.0, A 0, B 90, C 0} C_DIS
LIN {X -20.72, Y -56.31, Z 84.0, A 0, B 90, C 0} C_DIS
LIN {X -18.39, Y -57.08, Z 84.0, A 0, B 90, C 0} C_DIS
LIN {X -17.07, Y -57.52, Z 84.0, A 0, B 90, C 0} C_DIS
LIN {X -14.69, Y -58.14, Z 84.0, A 0, B 90, C 0} C_DIS
LIN {X -13.35, Y -58.5, Z 84.0, A 0, B 90, C 0} C_DIS
LIN {X -10.94, Y -58.97, Z 84.0, A 0, B 90, C 0} C_DIS
LIN {X -9.58, Y -59.23, Z 84.0, A 0, B 90, C 0} C_DIS
LIN {X -7.13, Y -59.55, Z 84.0, A 0, B 90, C 0} C_DIS
LIN {X -5.76, Y -59.72, Z 84.0, A 0, B 90, C 0} C_DIS
LIN {X -3.3, Y -59.88, Z 84.0, A 0, B 90, C 0} C_DIS
LIN {X -1.92, Y -59.97, Z 84.0, A 0, B 90, C 0} C_DIS
LIN {X 0.54, Y -59.97, Z 84.0, A 0, B 90, C 0} C_DIS
LIN {X 1.92, Y -59.97, Z 84.0, A 0, B 90, C 0} C_DIS
LIN {X 4.38, Y -59.81, Z 84.0, A 0, B 90, C 0} C_DIS
LIN {X 5.76, Y -59.72, Z 84.0, A 0, B 90, C 0} C_DIS
LIN {X 8.2, Y -59.41, Z 84.0, A 0, B 90, C 0} C_DIS
LIN {X 9.58, Y -59.23, Z 84.0, A 0, B 90, C 0} C_DIS
LIN {X 11.99, Y -58.76, Z 84.0, A 0, B 90, C 0} C_DIS
LIN {X 13.35, Y -58.5, Z 84.0, A 0, B 90, C 0} C_DIS
LIN {X 15.73, Y -57.87, Z 84.0, A 0, B 90, C 0} C_DIS
LIN {X 17.07, Y -57.52, Z 84.0, A 0, B 90, C 0} C_DIS
LIN {X 19.41, Y -56.74, Z 84.0, A 0, B 90, C 0} C_DIS
LIN {X 20.72, Y -56.31, Z 84.0, A 0, B 90, C 0} C_DIS
LIN {X 23.0, Y -55.38, Z 84.0, A 0, B 90, C 0} C_DIS
LIN {X 24.29, Y -54.86, Z 84.0, A 0, B 90, C 0} C_DIS
LIN {X 26.5, Y -53.8, Z 84.0, A 0, B 90, C 0} C_DIS
LIN {X 27.75, Y -53.2, Z 84.0, A 0, B 90, C 0} C_DIS
LIN {X 29.9, Y -51.99, Z 84.0, A 0, B 90, C 0} C_DIS
LIN {X 31.1, Y -51.31, Z 84.0, A 0, B 90, C 0} C_DIS
LIN {X 33.17, Y -49.97, Z 84.0, A 0, B 90, C 0} C_DIS
LIN {X 34.33, Y -49.21, Z 84.0, A 0, B 90, C 0} C_DIS
LIN {X 36.3, Y -47.74, Z 84.0, A 0, B 90, C 0} C_DIS
LIN {X 37.41, Y -46.91, Z 84.0, A 0, B 90, C 0} C_DIS
LIN {X 39.28, Y -45.31, Z 84.0, A 0, B 90, C 0} C_DIS
LIN {X 40.34, Y -44.42, Z 84.0, A 0, B 90, C 0} C_DIS
LIN {X 42.11, Y -42.7, Z 84.0, A 0, B 90, C 0} C_DIS
LIN {X 43.1, Y -41.74, Z 84.0, A 0, B 90, C 0} C_DIS
LIN {X 44.76, Y -39.92, Z 84.0, A 0, B 90, C 0} C_DIS
LIN {X 45.69, Y -38.89, Z 84.0, A 0, B 90, C 0} C_DIS
LIN {X 47.22, Y -36.97, Z 84.0, A 0, B 90, C 0} C_DIS
LIN {X 48.08, Y -35.89, Z 84.0, A 0, B 90, C 0} C_DIS
LIN {X 49.49, Y -33.87, Z 84.0, A 0, B 90, C 0} C_DIS
LIN {X 50.29, Y -32.73, Z 84.0, A 0, B 90, C 0} C_DIS
LIN {X 51.56, Y -30.63, Z 84.0, A 0, B 90, C 0} C_DIS
LIN {X 52.28, Y -29.44, Z 84.0, A 0, B 90, C 0} C_DIS
LIN {X 53.42, Y -27.26, Z 84.0, A 0, B 90, C 0} C_DIS
LIN {X 54.06, Y -26.03, Z 84.0, A 0, B 90, C 0} C_DIS
LIN {X 55.05, Y -23.78, Z 84.0, A 0, B 90, C 0} C_DIS
LIN {X 55.62, Y -22.52, Z 84.0, A 0, B 90, C 0} C_DIS
LIN {X 56.47, Y -20.21, Z 84.0, A 0, B 90, C 0} C_DIS
LIN {X 56.94, Y -18.91, Z 84.0, A 0, B 90, C 0} C_DIS
LIN {X 57.64, Y -16.55, Z 84.0, A 0, B 90, C 0} C_DIS
LIN {X 58.04, Y -15.22, Z 84.0, A 0, B 90, C 0} C_DIS
LIN {X 58.59, Y -12.82, Z 84.0, A 0, B 90, C 0} C_DIS
LIN {X 58.89, Y -11.47, Z 84.0, A 0, B 90, C 0} C_DIS
LIN {X 59.29, Y -9.04, Z 84.0, A 0, B 90, C 0} C_DIS
LIN {X 59.51, Y -7.67, Z 84.0, A 0, B 90, C 0} C_DIS
LIN {X 59.74, Y -5.22, Z 84.0, A 0, B 90, C 0} C_DIS
LIN {X 59.88, Y -3.84, Z 84.0, A 0, B 90, C 0} C_DIS
LIN {X 59.96, Y -1.38, Z 84.0, A 0, B 90, C 0} C_DIS
LIN {X 60.0, Y -0.0, Z 84.0, A 0, B 90, C 0} C_DIS
LIN {X 59.92, Y 2.46, Z 84.0, A 0, B 90, C 0} C_DIS
LIN {X 59.88, Y 3.84, Z 84.0, A 0, B 90, C 0} C_DIS
LIN {X 59.64, Y 6.29, Z 84.0, A 0, B 90, C 0} C_DIS
LIN {X 59.51, Y 7.67, Z 84.0, A 0, B 90, C 0} C_DIS
LIN {X 59.11, Y 10.1, Z 84.0, A 0, B 90, C 0} C_DIS
LIN {X 58.89, Y 11.47, Z 84.0, A 0, B 90, C 0} C_DIS
LIN {X 58.35, Y 13.87, Z 84.0, A 0, B 90, C 0} C_DIS
LIN {X 58.04, Y 15.22, Z 84.0, A 0, B 90, C 0} C_DIS
LIN {X 57.34, Y 17.58, Z 84.0, A 0, B 90, C 0} C_DIS
LIN {X 56.94, Y 18.91, Z 84.0, A 0, B 90, C 0} C_DIS
LIN {X 56.09, Y 21.22, Z 84.0, A 0, B 90, C 0} C_DIS
LIN {X 55.62, Y 22.52, Z 84.0, A 0, B 90, C 0} C_DIS
LIN {X 54.62, Y 24.77, Z 84.0, A 0, B 90, C 0} C_DIS
LIN {X 54.06, Y 26.03, Z 84.0, A 0, B 90, C 0} C_DIS
LIN {X 52.92, Y 28.22, Z 84.0, A 0, B 90, C 0} C_DIS
LIN {X 52.28, Y 29.44, Z 84.0, A 0, B 90, C 0} C_DIS
LIN {X 51.0, Y 31.55, Z 84.0, A 0, B 90, C 0} C_DIS
LIN {X 50.29, Y 32.73, Z 84.0, A 0, B 90, C 0} C_DIS
LIN {X 48.88, Y 34.75, Z 84.0, A 0, B 90, C 0} C_DIS
LIN {X 48.08, Y 35.89, Z 84.0, A 0, B 90, C 0} C_DIS
LIN {X 46.55, Y 37.81, Z 84.0, A 0, B 90, C 0} C_DIS
LIN {X 45.69, Y 38.89, Z 84.0, A 0, B 90, C 0} C_DIS
LIN {X 44.03, Y 40.72, Z 84.0, A 0, B 90, C 0} C_DIS
LIN {X 43.1, Y 41.74, Z 84.0, A 0, B 90, C 0} C_DIS
LIN {X 41.33, Y 43.45, Z 84.0, A 0, B 90, C 0} C_DIS
LIN {X 40.34, Y 44.42, Z 84.0, A 0, B 90, C 0} C_DIS
LIN {X 38.46, Y 46.01, Z 84.0, A 0, B 90, C 0} C_DIS
LIN {X 37.41, Y 46.91, Z 84.0, A 0, B 90, C 0} C_DIS
LIN {X 35.44, Y 48.38, Z 84.0, A 0, B 90, C 0} C_DIS
LIN {X 34.33, Y 49.21, Z 84.0, A 0, B 90, C 0} C_DIS
LIN {X 32.26, Y 50.55, Z 84.0, A 0, B 90, C 0} C_DIS
LIN {X 31.1, Y 51.31, Z 84.0, A 0, B 90, C 0} C_DIS
LIN {X 28.96, Y 52.52, Z 84.0, A 0, B 90, C 0} C_DIS
LIN {X 27.75, Y 53.2, Z 84.0, A 0, B 90, C 0} C_DIS
LIN {X 25.53, Y 54.26, Z 84.0, A 0, B 90, C 0} C_DIS
LIN {X 24.29, Y 54.86, Z 84.0, A 0, B 90, C 0} C_DIS
LIN {X 22.01, Y 55.79, Z 84.0, A 0, B 90, C 0} C_DIS
LIN {X 20.72, Y 56.31, Z 84.0, A 0, B 90, C 0} C_DIS
LIN {X 18.39, Y 57.08, Z 84.0, A 0, B 90, C 0} C_DIS
LIN {X 17.07, Y 57.52, Z 84.0, A 0, B 90, C 0} C_DIS
LIN {X 14.69, Y 58.14, Z 84.0, A 0, B 90, C 0} C_DIS
LIN {X 13.35, Y 58.5, Z 84.0, A 0, B 90, C 0} C_DIS
LIN {X 10.94, Y 58.97, Z 84.0, A 0, B 90, C 0} C_DIS
LIN {X 9.58, Y 59.23, Z 84.0, A 0, B 90, C 0} C_DIS
LIN {X 7.13, Y 59.55, Z 84.0, A 0, B 90, C 0} C_DIS
LIN {X 5.76, Y 59.72, Z 84.0, A 0, B 90, C 0} C_DIS
LIN {X 3.3, Y 59.88, Z 84.0, A 0, B 90, C 0} C_DIS
LIN {X 1.92, Y 59.97, Z 84.0, A 0, B 90, C 0} C_DIS
LIN {X -0.54, Y 59.97, Z 84.0, A 0, B 90, C 0} C_DIS
LIN {X -1.92, Y 59.97, Z 84.0, A 0, B 90, C 0} C_DIS
LIN {X -4.38, Y 59.81, Z 84.0, A 0, B 90, C 0} C_DIS
LIN {X -5.76, Y 59.72, Z 84.0, A 0, B 90, C 0} C_DIS
LIN {X -8.2, Y 59.41, Z 84.0, A 0, B 90, C 0} C_DIS
LIN {X -9.58, Y 59.23, Z 84.0, A 0, B 90, C 0} C_DIS
LIN {X -11.99, Y 58.76, Z 84.0, A 0, B 90, C 0} C_DIS
LIN {X -13.35, Y 58.5, Z 84.0, A 0, B 90, C 0} C_DIS
LIN {X -15.73, Y 57.87, Z 84.0, A 0, B 90, C 0} C_DIS
LIN {X -17.07, Y 57.52, Z 84.0, A 0, B 90, C 0} C_DIS
LIN {X -19.41, Y 56.74, Z 84.0, A 0, B 90, C 0} C_DIS
LIN {X -20.72, Y 56.31, Z 84.0, A 0, B 90, C 0} C_DIS
LIN {X -23.0, Y 55.38, Z 84.0, A 0, B 90, C 0} C_DIS
LIN {X -24.29, Y 54.86, Z 84.0, A 0, B 90, C 0} C_DIS
LIN {X -26.5, Y 53.8, Z 84.0, A 0, B 90, C 0} C_DIS
LIN {X -27.75, Y 53.2, Z 84.0, A 0, B 90, C 0} C_DIS
LIN {X -29.9, Y 51.99, Z 84.0, A 0, B 90, C 0} C_DIS
LIN {X -31.1, Y 51.31, Z 84.0, A 0, B 90, C 0} C_DIS
LIN {X -33.17, Y 49.97, Z 84.0, A 0, B 90, C 0} C_DIS
LIN {X -34.33, Y 49.21, Z 84.0, A 0, B 90, C 0} C_DIS
LIN {X -36.3, Y 47.74, Z 84.0, A 0, B 90, C 0} C_DIS
LIN {X -37.41, Y 46.91, Z 84.0, A 0, B 90, C 0} C_DIS
LIN {X -39.28, Y 45.31, Z 84.0, A 0, B 90, C 0} C_DIS
LIN {X -40.34, Y 44.42, Z 84.0, A 0, B 90, C 0} C_DIS
LIN {X -42.11, Y 42.7, Z 84.0, A 0, B 90, C 0} C_DIS
LIN {X -43.1, Y 41.74, Z 84.0, A 0, B 90, C 0} C_DIS
LIN {X -44.76, Y 39.92, Z 84.0, A 0, B 90, C 0} C_DIS
LIN {X -45.69, Y 38.89, Z 84.0, A 0, B 90, C 0} C_DIS
LIN {X -47.22, Y 36.97, Z 84.0, A 0, B 90, C 0} C_DIS
LIN {X -48.08, Y 35.89, Z 84.0, A 0, B 90, C 0} C_DIS
LIN {X -49.49, Y 33.87, Z 84.0, A 0, B 90, C 0} C_DIS
LIN {X -50.29, Y 32.73, Z 84.0, A 0, B 90, C 0} C_DIS
LIN {X -51.56, Y 30.63, Z 84.0, A 0, B 90, C 0} C_DIS
LIN {X -52.28, Y 29.44, Z 84.0, A 0, B 90, C 0} C_DIS
LIN {X -53.42, Y 27.26, Z 84.0, A 0, B 90, C 0} C_DIS
LIN {X -54.06, Y 26.03, Z 84.0, A 0, B 90, C 0} C_DIS
LIN {X -55.05, Y 23.78, Z 84.0, A 0, B 90, C 0} C_DIS
LIN {X -55.62, Y 22.52, Z 84.0, A 0, B 90, C 0} C_DIS
LIN {X -56.47, Y 20.21, Z 84.0, A 0, B 90, C 0} C_DIS
LIN {X -56.94, Y 18.91, Z 84.0, A 0, B 90, C 0} C_DIS
LIN {X -57.64, Y 16.55, Z 84.0, A 0, B 90, C 0} C_DIS
LIN {X -58.04, Y 15.22, Z 84.0, A 0, B 90, C 0} C_DIS
LIN {X -58.59, Y 12.82, Z 84.0, A 0, B 90, C 0} C_DIS
LIN {X -58.89, Y 11.47, Z 84.0, A 0, B 90, C 0} C_DIS
LIN {X -59.29, Y 9.04, Z 84.0, A 0, B 90, C 0} C_DIS
LIN {X -59.51, Y 7.67, Z 84.0, A 0, B 90, C 0} C_DIS
LIN {X -59.74, Y 5.22, Z 84.0, A 0, B 90, C 0} C_DIS
LIN {X -59.88, Y 3.84, Z 84.0, A 0, B 90, C 0} C_DIS
LIN {X -59.96, Y 1.38, Z 84.0, A 0, B 90, C 0} C_DIS
LIN {X -60.0, Y -0.0, Z 84.0, A 0, B 90, C 0} C_DIS
LIN {X -59.92, Y -2.46, Z 84.0, A 0, B 90, C 0} C_DIS
LIN {X -59.88, Y -3.84, Z 84.0, A 0, B 90, C 0} C_DIS
LIN {X -59.64, Y -6.29, Z 84.0, A 0, B 90, C 0} C_DIS
LIN {X -59.51, Y -7.67, Z 84.0, A 0, B 90, C 0} C_DIS
LIN {X -59.11, Y -10.1, Z 84.0, A 0, B 90, C 0} C_DIS
LIN {X -58.89, Y -11.47, Z 84.0, A 0, B 90, C 0} C_DIS
LIN {X -58.35, Y -13.87, Z 84.0, A 0, B 90, C 0} C_DIS
LIN {X -58.04, Y -15.22, Z 84.0, A 0, B 90, C 0} C_DIS
LIN {X -57.34, Y -17.58, Z 84.0, A 0, B 90, C 0} C_DIS
LIN {X -56.94, Y -18.91, Z 84.0, A 0, B 90, C 0} C_DIS
LIN {X -56.09, Y -21.22, Z 84.0, A 0, B 90, C 0} C_DIS
LIN {X -55.62, Y -22.52, Z 84.0, A 0, B 90, C 0} C_DIS
LIN {X -54.62, Y -24.77, Z 84.0, A 0, B 90, C 0} C_DIS
LIN {X -54.06, Y -26.03, Z 84.0, A 0, B 90, C 0} C_DIS
LIN {X -52.92, Y -28.22, Z 84.0, A 0, B 90, C 0} C_DIS
LIN {X -52.28, Y -29.44, Z 84.0, A 0, B 90, C 0} C_DIS
LIN {X -51.0, Y -31.55, Z 84.0, A 0, B 90, C 0} C_DIS
LIN {X -50.29, Y -32.73, Z 84.0, A 0, B 90, C 0} C_DIS
LIN {X -48.88, Y -34.75, Z 84.0, A 0, B 90, C 0} C_DIS
LIN {X -48.08, Y -35.89, Z 84.0, A 0, B 90, C 0} C_DIS
LIN {X -46.55, Y -37.81, Z 84.0, A 0, B 90, C 0} C_DIS
LIN {X -45.69, Y -38.89, Z 84.0, A 0, B 90, C 0} C_DIS
LIN {X -44.03, Y -40.72, Z 84.0, A 0, B 90, C 0} C_DIS
LIN {X -43.1, Y -41.74, Z 84.0, A 0, B 90, C 0} C_DIS
LIN {X -41.33, Y -43.45, Z 84.0, A 0, B 90, C 0} C_DIS
LIN {X -40.34, Y -44.42, Z 84.0, A 0, B 90, C 0} C_DIS
LIN {X -38.46, Y -46.01, Z 84.0, A 0, B 90, C 0} C_DIS
LIN {X -37.41, Y -46.91, Z 84.0, A 0, B 90, C 0} C_DIS
LIN {X -35.44, Y -48.38, Z 84.0, A 0, B 90, C 0} C_DIS
$OUT[1] = FALSE

; END LAYER 41
LIN {X -34.33, Y -49.21, Z 84.0, A 0, B 90, C 0} C_DIS
WAIT SEC 3
LIN {X -34.33, Y -49.21, Z 86.0, A 0, B 90, C 0} C_DIS
$OUT[1] = TRUE
WAIT SEC 0.8
LIN {X -34.33, Y -49.21, Z 86.0, A 0, B 90, C 0} C_DIS
LIN {X -34.33, Y -49.21, Z 86.0, A 0, B 90, C 0} C_DIS
LIN {X -32.14, Y -50.64, Z 86.0, A 0, B 90, C 0} C_DIS
LIN {X -31.1, Y -51.31, Z 86.0, A 0, B 90, C 0} C_DIS
LIN {X -28.82, Y -52.59, Z 86.0, A 0, B 90, C 0} C_DIS
LIN {X -27.75, Y -53.2, Z 86.0, A 0, B 90, C 0} C_DIS
LIN {X -25.4, Y -54.33, Z 86.0, A 0, B 90, C 0} C_DIS
LIN {X -24.29, Y -54.86, Z 86.0, A 0, B 90, C 0} C_DIS
LIN {X -21.86, Y -55.85, Z 86.0, A 0, B 90, C 0} C_DIS
LIN {X -20.72, Y -56.31, Z 86.0, A 0, B 90, C 0} C_DIS
LIN {X -18.24, Y -57.13, Z 86.0, A 0, B 90, C 0} C_DIS
LIN {X -17.07, Y -57.52, Z 86.0, A 0, B 90, C 0} C_DIS
LIN {X -14.54, Y -58.18, Z 86.0, A 0, B 90, C 0} C_DIS
LIN {X -13.35, Y -58.5, Z 86.0, A 0, B 90, C 0} C_DIS
LIN {X -10.78, Y -59.0, Z 86.0, A 0, B 90, C 0} C_DIS
LIN {X -9.58, Y -59.23, Z 86.0, A 0, B 90, C 0} C_DIS
LIN {X -6.98, Y -59.57, Z 86.0, A 0, B 90, C 0} C_DIS
LIN {X -5.76, Y -59.72, Z 86.0, A 0, B 90, C 0} C_DIS
LIN {X -3.15, Y -59.89, Z 86.0, A 0, B 90, C 0} C_DIS
LIN {X -1.92, Y -59.97, Z 86.0, A 0, B 90, C 0} C_DIS
LIN {X 0.69, Y -59.97, Z 86.0, A 0, B 90, C 0} C_DIS
LIN {X 1.92, Y -59.97, Z 86.0, A 0, B 90, C 0} C_DIS
LIN {X 4.53, Y -59.8, Z 86.0, A 0, B 90, C 0} C_DIS
LIN {X 5.76, Y -59.72, Z 86.0, A 0, B 90, C 0} C_DIS
LIN {X 8.36, Y -59.39, Z 86.0, A 0, B 90, C 0} C_DIS
LIN {X 9.58, Y -59.23, Z 86.0, A 0, B 90, C 0} C_DIS
LIN {X 12.14, Y -58.73, Z 86.0, A 0, B 90, C 0} C_DIS
LIN {X 13.35, Y -58.5, Z 86.0, A 0, B 90, C 0} C_DIS
LIN {X 15.88, Y -57.83, Z 86.0, A 0, B 90, C 0} C_DIS
LIN {X 17.07, Y -57.52, Z 86.0, A 0, B 90, C 0} C_DIS
LIN {X 19.55, Y -56.7, Z 86.0, A 0, B 90, C 0} C_DIS
LIN {X 20.72, Y -56.31, Z 86.0, A 0, B 90, C 0} C_DIS
LIN {X 23.15, Y -55.33, Z 86.0, A 0, B 90, C 0} C_DIS
LIN {X 24.29, Y -54.86, Z 86.0, A 0, B 90, C 0} C_DIS
LIN {X 26.64, Y -53.73, Z 86.0, A 0, B 90, C 0} C_DIS
LIN {X 27.75, Y -53.2, Z 86.0, A 0, B 90, C 0} C_DIS
LIN {X 30.03, Y -51.91, Z 86.0, A 0, B 90, C 0} C_DIS
LIN {X 31.1, Y -51.31, Z 86.0, A 0, B 90, C 0} C_DIS
LIN {X 33.3, Y -49.88, Z 86.0, A 0, B 90, C 0} C_DIS
LIN {X 34.33, Y -49.21, Z 86.0, A 0, B 90, C 0} C_DIS
LIN {X 36.42, Y -47.65, Z 86.0, A 0, B 90, C 0} C_DIS
LIN {X 37.41, Y -46.91, Z 86.0, A 0, B 90, C 0} C_DIS
LIN {X 39.4, Y -45.21, Z 86.0, A 0, B 90, C 0} C_DIS
LIN {X 40.34, Y -44.42, Z 86.0, A 0, B 90, C 0} C_DIS
LIN {X 42.22, Y -42.6, Z 86.0, A 0, B 90, C 0} C_DIS
LIN {X 43.1, Y -41.74, Z 86.0, A 0, B 90, C 0} C_DIS
LIN {X 44.86, Y -39.8, Z 86.0, A 0, B 90, C 0} C_DIS
LIN {X 45.69, Y -38.89, Z 86.0, A 0, B 90, C 0} C_DIS
LIN {X 47.32, Y -36.85, Z 86.0, A 0, B 90, C 0} C_DIS
LIN {X 48.08, Y -35.89, Z 86.0, A 0, B 90, C 0} C_DIS
LIN {X 49.58, Y -33.74, Z 86.0, A 0, B 90, C 0} C_DIS
LIN {X 50.29, Y -32.73, Z 86.0, A 0, B 90, C 0} C_DIS
LIN {X 51.64, Y -30.5, Z 86.0, A 0, B 90, C 0} C_DIS
LIN {X 52.28, Y -29.44, Z 86.0, A 0, B 90, C 0} C_DIS
LIN {X 53.49, Y -27.12, Z 86.0, A 0, B 90, C 0} C_DIS
LIN {X 54.06, Y -26.03, Z 86.0, A 0, B 90, C 0} C_DIS
LIN {X 55.12, Y -23.64, Z 86.0, A 0, B 90, C 0} C_DIS
LIN {X 55.62, Y -22.52, Z 86.0, A 0, B 90, C 0} C_DIS
LIN {X 56.52, Y -20.06, Z 86.0, A 0, B 90, C 0} C_DIS
LIN {X 56.94, Y -18.91, Z 86.0, A 0, B 90, C 0} C_DIS
LIN {X 57.69, Y -16.4, Z 86.0, A 0, B 90, C 0} C_DIS
LIN {X 58.04, Y -15.22, Z 86.0, A 0, B 90, C 0} C_DIS
LIN {X 58.62, Y -12.67, Z 86.0, A 0, B 90, C 0} C_DIS
LIN {X 58.89, Y -11.47, Z 86.0, A 0, B 90, C 0} C_DIS
LIN {X 59.31, Y -8.89, Z 86.0, A 0, B 90, C 0} C_DIS
LIN {X 59.51, Y -7.67, Z 86.0, A 0, B 90, C 0} C_DIS
LIN {X 59.76, Y -5.07, Z 86.0, A 0, B 90, C 0} C_DIS
LIN {X 59.88, Y -3.84, Z 86.0, A 0, B 90, C 0} C_DIS
LIN {X 59.96, Y -1.23, Z 86.0, A 0, B 90, C 0} C_DIS
LIN {X 60.0, Y 0.0, Z 86.0, A 0, B 90, C 0} C_DIS
LIN {X 59.92, Y 2.61, Z 86.0, A 0, B 90, C 0} C_DIS
LIN {X 59.88, Y 3.84, Z 86.0, A 0, B 90, C 0} C_DIS
LIN {X 59.63, Y 6.45, Z 86.0, A 0, B 90, C 0} C_DIS
LIN {X 59.51, Y 7.67, Z 86.0, A 0, B 90, C 0} C_DIS
LIN {X 59.09, Y 10.25, Z 86.0, A 0, B 90, C 0} C_DIS
LIN {X 58.89, Y 11.47, Z 86.0, A 0, B 90, C 0} C_DIS
LIN {X 58.31, Y 14.02, Z 86.0, A 0, B 90, C 0} C_DIS
LIN {X 58.04, Y 15.22, Z 86.0, A 0, B 90, C 0} C_DIS
LIN {X 57.29, Y 17.73, Z 86.0, A 0, B 90, C 0} C_DIS
LIN {X 56.94, Y 18.91, Z 86.0, A 0, B 90, C 0} C_DIS
LIN {X 56.04, Y 21.36, Z 86.0, A 0, B 90, C 0} C_DIS
LIN {X 55.62, Y 22.52, Z 86.0, A 0, B 90, C 0} C_DIS
LIN {X 54.56, Y 24.91, Z 86.0, A 0, B 90, C 0} C_DIS
LIN {X 54.06, Y 26.03, Z 86.0, A 0, B 90, C 0} C_DIS
LIN {X 52.85, Y 28.35, Z 86.0, A 0, B 90, C 0} C_DIS
LIN {X 52.28, Y 29.44, Z 86.0, A 0, B 90, C 0} C_DIS
LIN {X 50.92, Y 31.68, Z 86.0, A 0, B 90, C 0} C_DIS
LIN {X 50.29, Y 32.73, Z 86.0, A 0, B 90, C 0} C_DIS
LIN {X 48.79, Y 34.88, Z 86.0, A 0, B 90, C 0} C_DIS
LIN {X 48.08, Y 35.89, Z 86.0, A 0, B 90, C 0} C_DIS
LIN {X 46.45, Y 37.93, Z 86.0, A 0, B 90, C 0} C_DIS
LIN {X 45.69, Y 38.89, Z 86.0, A 0, B 90, C 0} C_DIS
LIN {X 43.93, Y 40.83, Z 86.0, A 0, B 90, C 0} C_DIS
LIN {X 43.1, Y 41.74, Z 86.0, A 0, B 90, C 0} C_DIS
LIN {X 41.22, Y 43.56, Z 86.0, A 0, B 90, C 0} C_DIS
LIN {X 40.34, Y 44.42, Z 86.0, A 0, B 90, C 0} C_DIS
LIN {X 38.35, Y 46.11, Z 86.0, A 0, B 90, C 0} C_DIS
LIN {X 37.41, Y 46.91, Z 86.0, A 0, B 90, C 0} C_DIS
LIN {X 35.31, Y 48.47, Z 86.0, A 0, B 90, C 0} C_DIS
LIN {X 34.33, Y 49.21, Z 86.0, A 0, B 90, C 0} C_DIS
LIN {X 32.14, Y 50.64, Z 86.0, A 0, B 90, C 0} C_DIS
LIN {X 31.1, Y 51.31, Z 86.0, A 0, B 90, C 0} C_DIS
LIN {X 28.82, Y 52.59, Z 86.0, A 0, B 90, C 0} C_DIS
LIN {X 27.75, Y 53.2, Z 86.0, A 0, B 90, C 0} C_DIS
LIN {X 25.4, Y 54.33, Z 86.0, A 0, B 90, C 0} C_DIS
LIN {X 24.29, Y 54.86, Z 86.0, A 0, B 90, C 0} C_DIS
LIN {X 21.86, Y 55.85, Z 86.0, A 0, B 90, C 0} C_DIS
LIN {X 20.72, Y 56.31, Z 86.0, A 0, B 90, C 0} C_DIS
LIN {X 18.24, Y 57.13, Z 86.0, A 0, B 90, C 0} C_DIS
LIN {X 17.07, Y 57.52, Z 86.0, A 0, B 90, C 0} C_DIS
LIN {X 14.54, Y 58.18, Z 86.0, A 0, B 90, C 0} C_DIS
LIN {X 13.35, Y 58.5, Z 86.0, A 0, B 90, C 0} C_DIS
LIN {X 10.78, Y 59.0, Z 86.0, A 0, B 90, C 0} C_DIS
LIN {X 9.58, Y 59.23, Z 86.0, A 0, B 90, C 0} C_DIS
LIN {X 6.98, Y 59.57, Z 86.0, A 0, B 90, C 0} C_DIS
LIN {X 5.76, Y 59.72, Z 86.0, A 0, B 90, C 0} C_DIS
LIN {X 3.15, Y 59.89, Z 86.0, A 0, B 90, C 0} C_DIS
LIN {X 1.92, Y 59.97, Z 86.0, A 0, B 90, C 0} C_DIS
LIN {X -0.69, Y 59.97, Z 86.0, A 0, B 90, C 0} C_DIS
LIN {X -1.92, Y 59.97, Z 86.0, A 0, B 90, C 0} C_DIS
LIN {X -4.53, Y 59.8, Z 86.0, A 0, B 90, C 0} C_DIS
LIN {X -5.76, Y 59.72, Z 86.0, A 0, B 90, C 0} C_DIS
LIN {X -8.36, Y 59.39, Z 86.0, A 0, B 90, C 0} C_DIS
LIN {X -9.58, Y 59.23, Z 86.0, A 0, B 90, C 0} C_DIS
LIN {X -12.14, Y 58.73, Z 86.0, A 0, B 90, C 0} C_DIS
LIN {X -13.35, Y 58.5, Z 86.0, A 0, B 90, C 0} C_DIS
LIN {X -15.88, Y 57.83, Z 86.0, A 0, B 90, C 0} C_DIS
LIN {X -17.07, Y 57.52, Z 86.0, A 0, B 90, C 0} C_DIS
LIN {X -19.55, Y 56.7, Z 86.0, A 0, B 90, C 0} C_DIS
LIN {X -20.72, Y 56.31, Z 86.0, A 0, B 90, C 0} C_DIS
LIN {X -23.15, Y 55.33, Z 86.0, A 0, B 90, C 0} C_DIS
LIN {X -24.29, Y 54.86, Z 86.0, A 0, B 90, C 0} C_DIS
LIN {X -26.64, Y 53.73, Z 86.0, A 0, B 90, C 0} C_DIS
LIN {X -27.75, Y 53.2, Z 86.0, A 0, B 90, C 0} C_DIS
LIN {X -30.03, Y 51.91, Z 86.0, A 0, B 90, C 0} C_DIS
LIN {X -31.1, Y 51.31, Z 86.0, A 0, B 90, C 0} C_DIS
LIN {X -33.3, Y 49.88, Z 86.0, A 0, B 90, C 0} C_DIS
LIN {X -34.33, Y 49.21, Z 86.0, A 0, B 90, C 0} C_DIS
LIN {X -36.42, Y 47.65, Z 86.0, A 0, B 90, C 0} C_DIS
LIN {X -37.41, Y 46.91, Z 86.0, A 0, B 90, C 0} C_DIS
LIN {X -39.4, Y 45.21, Z 86.0, A 0, B 90, C 0} C_DIS
LIN {X -40.34, Y 44.42, Z 86.0, A 0, B 90, C 0} C_DIS
LIN {X -42.22, Y 42.6, Z 86.0, A 0, B 90, C 0} C_DIS
LIN {X -43.1, Y 41.74, Z 86.0, A 0, B 90, C 0} C_DIS
LIN {X -44.86, Y 39.8, Z 86.0, A 0, B 90, C 0} C_DIS
LIN {X -45.69, Y 38.89, Z 86.0, A 0, B 90, C 0} C_DIS
LIN {X -47.32, Y 36.85, Z 86.0, A 0, B 90, C 0} C_DIS
LIN {X -48.08, Y 35.89, Z 86.0, A 0, B 90, C 0} C_DIS
LIN {X -49.58, Y 33.74, Z 86.0, A 0, B 90, C 0} C_DIS
LIN {X -50.29, Y 32.73, Z 86.0, A 0, B 90, C 0} C_DIS
LIN {X -51.64, Y 30.5, Z 86.0, A 0, B 90, C 0} C_DIS
LIN {X -52.28, Y 29.44, Z 86.0, A 0, B 90, C 0} C_DIS
LIN {X -53.49, Y 27.12, Z 86.0, A 0, B 90, C 0} C_DIS
LIN {X -54.06, Y 26.03, Z 86.0, A 0, B 90, C 0} C_DIS
LIN {X -55.12, Y 23.64, Z 86.0, A 0, B 90, C 0} C_DIS
LIN {X -55.62, Y 22.52, Z 86.0, A 0, B 90, C 0} C_DIS
LIN {X -56.52, Y 20.06, Z 86.0, A 0, B 90, C 0} C_DIS
LIN {X -56.94, Y 18.91, Z 86.0, A 0, B 90, C 0} C_DIS
LIN {X -57.69, Y 16.4, Z 86.0, A 0, B 90, C 0} C_DIS
LIN {X -58.04, Y 15.22, Z 86.0, A 0, B 90, C 0} C_DIS
LIN {X -58.62, Y 12.67, Z 86.0, A 0, B 90, C 0} C_DIS
LIN {X -58.89, Y 11.47, Z 86.0, A 0, B 90, C 0} C_DIS
LIN {X -59.31, Y 8.89, Z 86.0, A 0, B 90, C 0} C_DIS
LIN {X -59.51, Y 7.67, Z 86.0, A 0, B 90, C 0} C_DIS
LIN {X -59.76, Y 5.07, Z 86.0, A 0, B 90, C 0} C_DIS
LIN {X -59.88, Y 3.84, Z 86.0, A 0, B 90, C 0} C_DIS
LIN {X -59.96, Y 1.23, Z 86.0, A 0, B 90, C 0} C_DIS
LIN {X -60.0, Y -0.0, Z 86.0, A 0, B 90, C 0} C_DIS
LIN {X -59.92, Y -2.61, Z 86.0, A 0, B 90, C 0} C_DIS
LIN {X -59.88, Y -3.84, Z 86.0, A 0, B 90, C 0} C_DIS
LIN {X -59.63, Y -6.45, Z 86.0, A 0, B 90, C 0} C_DIS
LIN {X -59.51, Y -7.67, Z 86.0, A 0, B 90, C 0} C_DIS
LIN {X -59.09, Y -10.25, Z 86.0, A 0, B 90, C 0} C_DIS
LIN {X -58.89, Y -11.47, Z 86.0, A 0, B 90, C 0} C_DIS
LIN {X -58.31, Y -14.02, Z 86.0, A 0, B 90, C 0} C_DIS
LIN {X -58.04, Y -15.22, Z 86.0, A 0, B 90, C 0} C_DIS
LIN {X -57.29, Y -17.73, Z 86.0, A 0, B 90, C 0} C_DIS
LIN {X -56.94, Y -18.91, Z 86.0, A 0, B 90, C 0} C_DIS
LIN {X -56.04, Y -21.36, Z 86.0, A 0, B 90, C 0} C_DIS
LIN {X -55.62, Y -22.52, Z 86.0, A 0, B 90, C 0} C_DIS
LIN {X -54.56, Y -24.91, Z 86.0, A 0, B 90, C 0} C_DIS
LIN {X -54.06, Y -26.03, Z 86.0, A 0, B 90, C 0} C_DIS
LIN {X -52.85, Y -28.35, Z 86.0, A 0, B 90, C 0} C_DIS
LIN {X -52.28, Y -29.44, Z 86.0, A 0, B 90, C 0} C_DIS
LIN {X -50.92, Y -31.68, Z 86.0, A 0, B 90, C 0} C_DIS
LIN {X -50.29, Y -32.73, Z 86.0, A 0, B 90, C 0} C_DIS
LIN {X -48.79, Y -34.88, Z 86.0, A 0, B 90, C 0} C_DIS
LIN {X -48.08, Y -35.89, Z 86.0, A 0, B 90, C 0} C_DIS
LIN {X -46.45, Y -37.93, Z 86.0, A 0, B 90, C 0} C_DIS
LIN {X -45.69, Y -38.89, Z 86.0, A 0, B 90, C 0} C_DIS
LIN {X -43.93, Y -40.83, Z 86.0, A 0, B 90, C 0} C_DIS
LIN {X -43.1, Y -41.74, Z 86.0, A 0, B 90, C 0} C_DIS
LIN {X -41.22, Y -43.56, Z 86.0, A 0, B 90, C 0} C_DIS
LIN {X -40.34, Y -44.42, Z 86.0, A 0, B 90, C 0} C_DIS
LIN {X -38.35, Y -46.11, Z 86.0, A 0, B 90, C 0} C_DIS
LIN {X -37.41, Y -46.91, Z 86.0, A 0, B 90, C 0} C_DIS
LIN {X -35.31, Y -48.47, Z 86.0, A 0, B 90, C 0} C_DIS
$OUT[1] = FALSE

; END LAYER 42
LIN {X -34.33, Y -49.21, Z 86.0, A 0, B 90, C 0} C_DIS
WAIT SEC 3
LIN {X -34.33, Y -49.21, Z 88.0, A 0, B 90, C 0} C_DIS
$OUT[1] = TRUE
WAIT SEC 0.8
LIN {X -34.33, Y -49.21, Z 88.0, A 0, B 90, C 0} C_DIS
LIN {X -34.33, Y -49.21, Z 88.0, A 0, B 90, C 0} C_DIS
LIN {X -32.01, Y -50.72, Z 88.0, A 0, B 90, C 0} C_DIS
LIN {X -31.1, Y -51.31, Z 88.0, A 0, B 90, C 0} C_DIS
LIN {X -28.69, Y -52.67, Z 88.0, A 0, B 90, C 0} C_DIS
LIN {X -27.75, Y -53.2, Z 88.0, A 0, B 90, C 0} C_DIS
LIN {X -25.26, Y -54.4, Z 88.0, A 0, B 90, C 0} C_DIS
LIN {X -24.29, Y -54.86, Z 88.0, A 0, B 90, C 0} C_DIS
LIN {X -21.72, Y -55.9, Z 88.0, A 0, B 90, C 0} C_DIS
LIN {X -20.72, Y -56.31, Z 88.0, A 0, B 90, C 0} C_DIS
LIN {X -18.09, Y -57.18, Z 88.0, A 0, B 90, C 0} C_DIS
LIN {X -17.07, Y -57.52, Z 88.0, A 0, B 90, C 0} C_DIS
LIN {X -14.39, Y -58.22, Z 88.0, A 0, B 90, C 0} C_DIS
LIN {X -13.35, Y -58.5, Z 88.0, A 0, B 90, C 0} C_DIS
LIN {X -10.63, Y -59.03, Z 88.0, A 0, B 90, C 0} C_DIS
LIN {X -9.58, Y -59.23, Z 88.0, A 0, B 90, C 0} C_DIS
LIN {X -6.83, Y -59.59, Z 88.0, A 0, B 90, C 0} C_DIS
LIN {X -5.76, Y -59.72, Z 88.0, A 0, B 90, C 0} C_DIS
LIN {X -3.0, Y -59.9, Z 88.0, A 0, B 90, C 0} C_DIS
LIN {X -1.92, Y -59.97, Z 88.0, A 0, B 90, C 0} C_DIS
LIN {X 0.85, Y -59.97, Z 88.0, A 0, B 90, C 0} C_DIS
LIN {X 1.92, Y -59.97, Z 88.0, A 0, B 90, C 0} C_DIS
LIN {X 4.69, Y -59.79, Z 88.0, A 0, B 90, C 0} C_DIS
LIN {X 5.76, Y -59.72, Z 88.0, A 0, B 90, C 0} C_DIS
LIN {X 8.51, Y -59.37, Z 88.0, A 0, B 90, C 0} C_DIS
LIN {X 9.58, Y -59.23, Z 88.0, A 0, B 90, C 0} C_DIS
LIN {X 12.29, Y -58.7, Z 88.0, A 0, B 90, C 0} C_DIS
LIN {X 13.35, Y -58.5, Z 88.0, A 0, B 90, C 0} C_DIS
LIN {X 16.03, Y -57.79, Z 88.0, A 0, B 90, C 0} C_DIS
LIN {X 17.07, Y -57.52, Z 88.0, A 0, B 90, C 0} C_DIS
LIN {X 19.7, Y -56.65, Z 88.0, A 0, B 90, C 0} C_DIS
LIN {X 20.72, Y -56.31, Z 88.0, A 0, B 90, C 0} C_DIS
LIN {X 23.29, Y -55.27, Z 88.0, A 0, B 90, C 0} C_DIS
LIN {X 24.29, Y -54.86, Z 88.0, A 0, B 90, C 0} C_DIS
LIN {X 26.78, Y -53.66, Z 88.0, A 0, B 90, C 0} C_DIS
LIN {X 27.75, Y -53.2, Z 88.0, A 0, B 90, C 0} C_DIS
LIN {X 30.17, Y -51.84, Z 88.0, A 0, B 90, C 0} C_DIS
LIN {X 31.1, Y -51.31, Z 88.0, A 0, B 90, C 0} C_DIS
LIN {X 33.42, Y -49.8, Z 88.0, A 0, B 90, C 0} C_DIS
LIN {X 34.33, Y -49.21, Z 88.0, A 0, B 90, C 0} C_DIS
LIN {X 36.55, Y -47.55, Z 88.0, A 0, B 90, C 0} C_DIS
LIN {X 37.41, Y -46.91, Z 88.0, A 0, B 90, C 0} C_DIS
LIN {X 39.52, Y -45.11, Z 88.0, A 0, B 90, C 0} C_DIS
LIN {X 40.34, Y -44.42, Z 88.0, A 0, B 90, C 0} C_DIS
LIN {X 42.33, Y -42.49, Z 88.0, A 0, B 90, C 0} C_DIS
LIN {X 43.1, Y -41.74, Z 88.0, A 0, B 90, C 0} C_DIS
LIN {X 44.96, Y -39.69, Z 88.0, A 0, B 90, C 0} C_DIS
LIN {X 45.69, Y -38.89, Z 88.0, A 0, B 90, C 0} C_DIS
LIN {X 47.41, Y -36.73, Z 88.0, A 0, B 90, C 0} C_DIS
LIN {X 48.08, Y -35.89, Z 88.0, A 0, B 90, C 0} C_DIS
LIN {X 49.67, Y -33.62, Z 88.0, A 0, B 90, C 0} C_DIS
LIN {X 50.29, Y -32.73, Z 88.0, A 0, B 90, C 0} C_DIS
LIN {X 51.72, Y -30.36, Z 88.0, A 0, B 90, C 0} C_DIS
LIN {X 52.28, Y -29.44, Z 88.0, A 0, B 90, C 0} C_DIS
LIN {X 53.56, Y -26.99, Z 88.0, A 0, B 90, C 0} C_DIS
LIN {X 54.06, Y -26.03, Z 88.0, A 0, B 90, C 0} C_DIS
LIN {X 55.18, Y -23.5, Z 88.0, A 0, B 90, C 0} C_DIS
LIN {X 55.62, Y -22.52, Z 88.0, A 0, B 90, C 0} C_DIS
LIN {X 56.57, Y -19.92, Z 88.0, A 0, B 90, C 0} C_DIS
LIN {X 56.94, Y -18.91, Z 88.0, A 0, B 90, C 0} C_DIS
LIN {X 57.73, Y -16.25, Z 88.0, A 0, B 90, C 0} C_DIS
LIN {X 58.04, Y -15.22, Z 88.0, A 0, B 90, C 0} C_DIS
LIN {X 58.65, Y -12.52, Z 88.0, A 0, B 90, C 0} C_DIS
LIN {X 58.89, Y -11.47, Z 88.0, A 0, B 90, C 0} C_DIS
LIN {X 59.34, Y -8.74, Z 88.0, A 0, B 90, C 0} C_DIS
LIN {X 59.51, Y -7.67, Z 88.0, A 0, B 90, C 0} C_DIS
LIN {X 59.77, Y -4.92, Z 88.0, A 0, B 90, C 0} C_DIS
LIN {X 59.88, Y -3.84, Z 88.0, A 0, B 90, C 0} C_DIS
LIN {X 59.97, Y -1.08, Z 88.0, A 0, B 90, C 0} C_DIS
LIN {X 60.0, Y 0.0, Z 88.0, A 0, B 90, C 0} C_DIS
LIN {X 59.91, Y 2.77, Z 88.0, A 0, B 90, C 0} C_DIS
LIN {X 59.88, Y 3.84, Z 88.0, A 0, B 90, C 0} C_DIS
LIN {X 59.61, Y 6.6, Z 88.0, A 0, B 90, C 0} C_DIS
LIN {X 59.51, Y 7.67, Z 88.0, A 0, B 90, C 0} C_DIS
LIN {X 59.07, Y 10.41, Z 88.0, A 0, B 90, C 0} C_DIS
LIN {X 58.89, Y 11.47, Z 88.0, A 0, B 90, C 0} C_DIS
LIN {X 58.28, Y 14.17, Z 88.0, A 0, B 90, C 0} C_DIS
LIN {X 58.04, Y 15.22, Z 88.0, A 0, B 90, C 0} C_DIS
LIN {X 57.25, Y 17.87, Z 88.0, A 0, B 90, C 0} C_DIS
LIN {X 56.94, Y 18.91, Z 88.0, A 0, B 90, C 0} C_DIS
LIN {X 55.99, Y 21.51, Z 88.0, A 0, B 90, C 0} C_DIS
LIN {X 55.62, Y 22.52, Z 88.0, A 0, B 90, C 0} C_DIS
LIN {X 54.49, Y 25.05, Z 88.0, A 0, B 90, C 0} C_DIS
LIN {X 54.06, Y 26.03, Z 88.0, A 0, B 90, C 0} C_DIS
LIN {X 52.78, Y 28.49, Z 88.0, A 0, B 90, C 0} C_DIS
LIN {X 52.28, Y 29.44, Z 88.0, A 0, B 90, C 0} C_DIS
LIN {X 50.84, Y 31.81, Z 88.0, A 0, B 90, C 0} C_DIS
LIN {X 50.29, Y 32.73, Z 88.0, A 0, B 90, C 0} C_DIS
LIN {X 48.7, Y 35.0, Z 88.0, A 0, B 90, C 0} C_DIS
LIN {X 48.08, Y 35.89, Z 88.0, A 0, B 90, C 0} C_DIS
LIN {X 46.36, Y 38.05, Z 88.0, A 0, B 90, C 0} C_DIS
LIN {X 45.69, Y 38.89, Z 88.0, A 0, B 90, C 0} C_DIS
LIN {X 43.82, Y 40.94, Z 88.0, A 0, B 90, C 0} C_DIS
LIN {X 43.1, Y 41.74, Z 88.0, A 0, B 90, C 0} C_DIS
LIN {X 41.11, Y 43.67, Z 88.0, A 0, B 90, C 0} C_DIS
LIN {X 40.34, Y 44.42, Z 88.0, A 0, B 90, C 0} C_DIS
LIN {X 38.23, Y 46.21, Z 88.0, A 0, B 90, C 0} C_DIS
LIN {X 37.41, Y 46.91, Z 88.0, A 0, B 90, C 0} C_DIS
LIN {X 35.19, Y 48.57, Z 88.0, A 0, B 90, C 0} C_DIS
LIN {X 34.33, Y 49.21, Z 88.0, A 0, B 90, C 0} C_DIS
LIN {X 32.01, Y 50.72, Z 88.0, A 0, B 90, C 0} C_DIS
LIN {X 31.1, Y 51.31, Z 88.0, A 0, B 90, C 0} C_DIS
LIN {X 28.69, Y 52.67, Z 88.0, A 0, B 90, C 0} C_DIS
LIN {X 27.75, Y 53.2, Z 88.0, A 0, B 90, C 0} C_DIS
LIN {X 25.26, Y 54.4, Z 88.0, A 0, B 90, C 0} C_DIS
LIN {X 24.29, Y 54.86, Z 88.0, A 0, B 90, C 0} C_DIS
LIN {X 21.72, Y 55.9, Z 88.0, A 0, B 90, C 0} C_DIS
LIN {X 20.72, Y 56.31, Z 88.0, A 0, B 90, C 0} C_DIS
LIN {X 18.09, Y 57.18, Z 88.0, A 0, B 90, C 0} C_DIS
LIN {X 17.07, Y 57.52, Z 88.0, A 0, B 90, C 0} C_DIS
LIN {X 14.39, Y 58.22, Z 88.0, A 0, B 90, C 0} C_DIS
LIN {X 13.35, Y 58.5, Z 88.0, A 0, B 90, C 0} C_DIS
LIN {X 10.63, Y 59.03, Z 88.0, A 0, B 90, C 0} C_DIS
LIN {X 9.58, Y 59.23, Z 88.0, A 0, B 90, C 0} C_DIS
LIN {X 6.83, Y 59.59, Z 88.0, A 0, B 90, C 0} C_DIS
LIN {X 5.76, Y 59.72, Z 88.0, A 0, B 90, C 0} C_DIS
LIN {X 3.0, Y 59.9, Z 88.0, A 0, B 90, C 0} C_DIS
LIN {X 1.92, Y 59.97, Z 88.0, A 0, B 90, C 0} C_DIS
LIN {X -0.85, Y 59.97, Z 88.0, A 0, B 90, C 0} C_DIS
LIN {X -1.92, Y 59.97, Z 88.0, A 0, B 90, C 0} C_DIS
LIN {X -4.69, Y 59.79, Z 88.0, A 0, B 90, C 0} C_DIS
LIN {X -5.76, Y 59.72, Z 88.0, A 0, B 90, C 0} C_DIS
LIN {X -8.51, Y 59.37, Z 88.0, A 0, B 90, C 0} C_DIS
LIN {X -9.58, Y 59.23, Z 88.0, A 0, B 90, C 0} C_DIS
LIN {X -12.29, Y 58.7, Z 88.0, A 0, B 90, C 0} C_DIS
LIN {X -13.35, Y 58.5, Z 88.0, A 0, B 90, C 0} C_DIS
LIN {X -16.03, Y 57.79, Z 88.0, A 0, B 90, C 0} C_DIS
LIN {X -17.07, Y 57.52, Z 88.0, A 0, B 90, C 0} C_DIS
LIN {X -19.7, Y 56.65, Z 88.0, A 0, B 90, C 0} C_DIS
LIN {X -20.72, Y 56.31, Z 88.0, A 0, B 90, C 0} C_DIS
LIN {X -23.29, Y 55.27, Z 88.0, A 0, B 90, C 0} C_DIS
LIN {X -24.29, Y 54.86, Z 88.0, A 0, B 90, C 0} C_DIS
LIN {X -26.78, Y 53.66, Z 88.0, A 0, B 90, C 0} C_DIS
LIN {X -27.75, Y 53.2, Z 88.0, A 0, B 90, C 0} C_DIS
LIN {X -30.17, Y 51.84, Z 88.0, A 0, B 90, C 0} C_DIS
LIN {X -31.1, Y 51.31, Z 88.0, A 0, B 90, C 0} C_DIS
LIN {X -33.42, Y 49.8, Z 88.0, A 0, B 90, C 0} C_DIS
LIN {X -34.33, Y 49.21, Z 88.0, A 0, B 90, C 0} C_DIS
LIN {X -36.55, Y 47.55, Z 88.0, A 0, B 90, C 0} C_DIS
LIN {X -37.41, Y 46.91, Z 88.0, A 0, B 90, C 0} C_DIS
LIN {X -39.52, Y 45.11, Z 88.0, A 0, B 90, C 0} C_DIS
LIN {X -40.34, Y 44.42, Z 88.0, A 0, B 90, C 0} C_DIS
LIN {X -42.33, Y 42.49, Z 88.0, A 0, B 90, C 0} C_DIS
LIN {X -43.1, Y 41.74, Z 88.0, A 0, B 90, C 0} C_DIS
LIN {X -44.96, Y 39.69, Z 88.0, A 0, B 90, C 0} C_DIS
LIN {X -45.69, Y 38.89, Z 88.0, A 0, B 90, C 0} C_DIS
LIN {X -47.41, Y 36.73, Z 88.0, A 0, B 90, C 0} C_DIS
LIN {X -48.08, Y 35.89, Z 88.0, A 0, B 90, C 0} C_DIS
LIN {X -49.67, Y 33.62, Z 88.0, A 0, B 90, C 0} C_DIS
LIN {X -50.29, Y 32.73, Z 88.0, A 0, B 90, C 0} C_DIS
LIN {X -51.72, Y 30.36, Z 88.0, A 0, B 90, C 0} C_DIS
LIN {X -52.28, Y 29.44, Z 88.0, A 0, B 90, C 0} C_DIS
LIN {X -53.56, Y 26.99, Z 88.0, A 0, B 90, C 0} C_DIS
LIN {X -54.06, Y 26.03, Z 88.0, A 0, B 90, C 0} C_DIS
LIN {X -55.18, Y 23.5, Z 88.0, A 0, B 90, C 0} C_DIS
LIN {X -55.62, Y 22.52, Z 88.0, A 0, B 90, C 0} C_DIS
LIN {X -56.57, Y 19.92, Z 88.0, A 0, B 90, C 0} C_DIS
LIN {X -56.94, Y 18.91, Z 88.0, A 0, B 90, C 0} C_DIS
LIN {X -57.73, Y 16.25, Z 88.0, A 0, B 90, C 0} C_DIS
LIN {X -58.04, Y 15.22, Z 88.0, A 0, B 90, C 0} C_DIS
LIN {X -58.65, Y 12.52, Z 88.0, A 0, B 90, C 0} C_DIS
LIN {X -58.89, Y 11.47, Z 88.0, A 0, B 90, C 0} C_DIS
LIN {X -59.34, Y 8.74, Z 88.0, A 0, B 90, C 0} C_DIS
LIN {X -59.51, Y 7.67, Z 88.0, A 0, B 90, C 0} C_DIS
LIN {X -59.77, Y 4.92, Z 88.0, A 0, B 90, C 0} C_DIS
LIN {X -59.88, Y 3.84, Z 88.0, A 0, B 90, C 0} C_DIS
LIN {X -59.97, Y 1.08, Z 88.0, A 0, B 90, C 0} C_DIS
LIN {X -60.0, Y -0.0, Z 88.0, A 0, B 90, C 0} C_DIS
LIN {X -59.91, Y -2.77, Z 88.0, A 0, B 90, C 0} C_DIS
LIN {X -59.88, Y -3.84, Z 88.0, A 0, B 90, C 0} C_DIS
LIN {X -59.61, Y -6.6, Z 88.0, A 0, B 90, C 0} C_DIS
LIN {X -59.51, Y -7.67, Z 88.0, A 0, B 90, C 0} C_DIS
LIN {X -59.07, Y -10.41, Z 88.0, A 0, B 90, C 0} C_DIS
LIN {X -58.89, Y -11.47, Z 88.0, A 0, B 90, C 0} C_DIS
LIN {X -58.28, Y -14.17, Z 88.0, A 0, B 90, C 0} C_DIS
LIN {X -58.04, Y -15.22, Z 88.0, A 0, B 90, C 0} C_DIS
LIN {X -57.25, Y -17.87, Z 88.0, A 0, B 90, C 0} C_DIS
LIN {X -56.94, Y -18.91, Z 88.0, A 0, B 90, C 0} C_DIS
LIN {X -55.99, Y -21.51, Z 88.0, A 0, B 90, C 0} C_DIS
LIN {X -55.62, Y -22.52, Z 88.0, A 0, B 90, C 0} C_DIS
LIN {X -54.49, Y -25.05, Z 88.0, A 0, B 90, C 0} C_DIS
LIN {X -54.06, Y -26.03, Z 88.0, A 0, B 90, C 0} C_DIS
LIN {X -52.78, Y -28.49, Z 88.0, A 0, B 90, C 0} C_DIS
LIN {X -52.28, Y -29.44, Z 88.0, A 0, B 90, C 0} C_DIS
LIN {X -50.84, Y -31.81, Z 88.0, A 0, B 90, C 0} C_DIS
LIN {X -50.29, Y -32.73, Z 88.0, A 0, B 90, C 0} C_DIS
LIN {X -48.7, Y -35.0, Z 88.0, A 0, B 90, C 0} C_DIS
LIN {X -48.08, Y -35.89, Z 88.0, A 0, B 90, C 0} C_DIS
LIN {X -46.36, Y -38.05, Z 88.0, A 0, B 90, C 0} C_DIS
LIN {X -45.69, Y -38.89, Z 88.0, A 0, B 90, C 0} C_DIS
LIN {X -43.82, Y -40.94, Z 88.0, A 0, B 90, C 0} C_DIS
LIN {X -43.1, Y -41.74, Z 88.0, A 0, B 90, C 0} C_DIS
LIN {X -41.11, Y -43.67, Z 88.0, A 0, B 90, C 0} C_DIS
LIN {X -40.34, Y -44.42, Z 88.0, A 0, B 90, C 0} C_DIS
LIN {X -38.23, Y -46.21, Z 88.0, A 0, B 90, C 0} C_DIS
LIN {X -37.41, Y -46.91, Z 88.0, A 0, B 90, C 0} C_DIS
LIN {X -35.19, Y -48.57, Z 88.0, A 0, B 90, C 0} C_DIS
$OUT[1] = FALSE

; END LAYER 43
LIN {X -34.33, Y -49.21, Z 88.0, A 0, B 90, C 0} C_DIS
WAIT SEC 3
LIN {X -34.33, Y -49.21, Z 90.0, A 0, B 90, C 0} C_DIS
$OUT[1] = TRUE
WAIT SEC 0.8
LIN {X -34.33, Y -49.21, Z 90.0, A 0, B 90, C 0} C_DIS
LIN {X -34.33, Y -49.21, Z 90.0, A 0, B 90, C 0} C_DIS
LIN {X -31.88, Y -50.8, Z 90.0, A 0, B 90, C 0} C_DIS
LIN {X -31.1, Y -51.31, Z 90.0, A 0, B 90, C 0} C_DIS
LIN {X -28.56, Y -52.74, Z 90.0, A 0, B 90, C 0} C_DIS
LIN {X -27.75, Y -53.2, Z 90.0, A 0, B 90, C 0} C_DIS
LIN {X -25.12, Y -54.46, Z 90.0, A 0, B 90, C 0} C_DIS
LIN {X -24.29, Y -54.86, Z 90.0, A 0, B 90, C 0} C_DIS
LIN {X -21.58, Y -55.96, Z 90.0, A 0, B 90, C 0} C_DIS
LIN {X -20.72, Y -56.31, Z 90.0, A 0, B 90, C 0} C_DIS
LIN {X -17.95, Y -57.23, Z 90.0, A 0, B 90, C 0} C_DIS
LIN {X -17.07, Y -57.52, Z 90.0, A 0, B 90, C 0} C_DIS
LIN {X -14.24, Y -58.26, Z 90.0, A 0, B 90, C 0} C_DIS
LIN {X -13.35, Y -58.5, Z 90.0, A 0, B 90, C 0} C_DIS
LIN {X -10.48, Y -59.05, Z 90.0, A 0, B 90, C 0} C_DIS
LIN {X -9.58, Y -59.23, Z 90.0, A 0, B 90, C 0} C_DIS
LIN {X -6.68, Y -59.6, Z 90.0, A 0, B 90, C 0} C_DIS
LIN {X -5.76, Y -59.72, Z 90.0, A 0, B 90, C 0} C_DIS
LIN {X -2.84, Y -59.91, Z 90.0, A 0, B 90, C 0} C_DIS
LIN {X -1.92, Y -59.97, Z 90.0, A 0, B 90, C 0} C_DIS
LIN {X 1.0, Y -59.97, Z 90.0, A 0, B 90, C 0} C_DIS
LIN {X 1.92, Y -59.97, Z 90.0, A 0, B 90, C 0} C_DIS
LIN {X 4.84, Y -59.78, Z 90.0, A 0, B 90, C 0} C_DIS
LIN {X 5.76, Y -59.72, Z 90.0, A 0, B 90, C 0} C_DIS
LIN {X 8.66, Y -59.35, Z 90.0, A 0, B 90, C 0} C_DIS
LIN {X 9.58, Y -59.23, Z 90.0, A 0, B 90, C 0} C_DIS
LIN {X 12.45, Y -58.67, Z 90.0, A 0, B 90, C 0} C_DIS
LIN {X 13.35, Y -58.5, Z 90.0, A 0, B 90, C 0} C_DIS
LIN {X 16.18, Y -57.75, Z 90.0, A 0, B 90, C 0} C_DIS
LIN {X 17.07, Y -57.52, Z 90.0, A 0, B 90, C 0} C_DIS
LIN {X 19.85, Y -56.6, Z 90.0, A 0, B 90, C 0} C_DIS
LIN {X 20.72, Y -56.31, Z 90.0, A 0, B 90, C 0} C_DIS
LIN {X 23.43, Y -55.21, Z 90.0, A 0, B 90, C 0} C_DIS
LIN {X 24.29, Y -54.86, Z 90.0, A 0, B 90, C 0} C_DIS
LIN {X 26.92, Y -53.6, Z 90.0, A 0, B 90, C 0} C_DIS
LIN {X 27.75, Y -53.2, Z 90.0, A 0, B 90, C 0} C_DIS
LIN {X 30.3, Y -51.76, Z 90.0, A 0, B 90, C 0} C_DIS
LIN {X 31.1, Y -51.31, Z 90.0, A 0, B 90, C 0} C_DIS
LIN {X 33.55, Y -49.71, Z 90.0, A 0, B 90, C 0} C_DIS
LIN {X 34.33, Y -49.21, Z 90.0, A 0, B 90, C 0} C_DIS
LIN {X 36.67, Y -47.46, Z 90.0, A 0, B 90, C 0} C_DIS
LIN {X 37.41, Y -46.91, Z 90.0, A 0, B 90, C 0} C_DIS
LIN {X 39.64, Y -45.02, Z 90.0, A 0, B 90, C 0} C_DIS
LIN {X 40.34, Y -44.42, Z 90.0, A 0, B 90, C 0} C_DIS
LIN {X 42.44, Y -42.38, Z 90.0, A 0, B 90, C 0} C_DIS
LIN {X 43.1, Y -41.74, Z 90.0, A 0, B 90, C 0} C_DIS
LIN {X 45.07, Y -39.58, Z 90.0, A 0, B 90, C 0} C_DIS
LIN {X 45.69, Y -38.89, Z 90.0, A 0, B 90, C 0} C_DIS
LIN {X 47.51, Y -36.61, Z 90.0, A 0, B 90, C 0} C_DIS
LIN {X 48.08, Y -35.89, Z 90.0, A 0, B 90, C 0} C_DIS
LIN {X 49.76, Y -33.49, Z 90.0, A 0, B 90, C 0} C_DIS
LIN {X 50.29, Y -32.73, Z 90.0, A 0, B 90, C 0} C_DIS
LIN {X 51.8, Y -30.23, Z 90.0, A 0, B 90, C 0} C_DIS
LIN {X 52.28, Y -29.44, Z 90.0, A 0, B 90, C 0} C_DIS
LIN {X 53.63, Y -26.85, Z 90.0, A 0, B 90, C 0} C_DIS
LIN {X 54.06, Y -26.03, Z 90.0, A 0, B 90, C 0} C_DIS
LIN {X 55.24, Y -23.36, Z 90.0, A 0, B 90, C 0} C_DIS
LIN {X 55.62, Y -22.52, Z 90.0, A 0, B 90, C 0} C_DIS
LIN {X 56.62, Y -19.77, Z 90.0, A 0, B 90, C 0} C_DIS
LIN {X 56.94, Y -18.91, Z 90.0, A 0, B 90, C 0} C_DIS
LIN {X 57.78, Y -16.1, Z 90.0, A 0, B 90, C 0} C_DIS
LIN {X 58.04, Y -15.22, Z 90.0, A 0, B 90, C 0} C_DIS
LIN {X 58.69, Y -12.37, Z 90.0, A 0, B 90, C 0} C_DIS
LIN {X 58.89, Y -11.47, Z 90.0, A 0, B 90, C 0} C_DIS
LIN {X 59.36, Y -8.58, Z 90.0, A 0, B 90, C 0} C_DIS
LIN {X 59.51, Y -7.67, Z 90.0, A 0, B 90, C 0} C_DIS
LIN {X 59.79, Y -4.76, Z 90.0, A 0, B 90, C 0} C_DIS
LIN {X 59.88, Y -3.84, Z 90.0, A 0, B 90, C 0} C_DIS
LIN {X 59.97, Y -0.92, Z 90.0, A 0, B 90, C 0} C_DIS
LIN {X 60.0, Y -0.0, Z 90.0, A 0, B 90, C 0} C_DIS
LIN {X 59.91, Y 2.92, Z 90.0, A 0, B 90, C 0} C_DIS
LIN {X 59.88, Y 3.84, Z 90.0, A 0, B 90, C 0} C_DIS
LIN {X 59.6, Y 6.75, Z 90.0, A 0, B 90, C 0} C_DIS
LIN {X 59.51, Y 7.67, Z 90.0, A 0, B 90, C 0} C_DIS
LIN {X 59.04, Y 10.56, Z 90.0, A 0, B 90, C 0} C_DIS
LIN {X 58.89, Y 11.47, Z 90.0, A 0, B 90, C 0} C_DIS
LIN {X 58.24, Y 14.32, Z 90.0, A 0, B 90, C 0} C_DIS
LIN {X 58.04, Y 15.22, Z 90.0, A 0, B 90, C 0} C_DIS
LIN {X 57.21, Y 18.02, Z 90.0, A 0, B 90, C 0} C_DIS
LIN {X 56.94, Y 18.91, Z 90.0, A 0, B 90, C 0} C_DIS
LIN {X 55.93, Y 21.65, Z 90.0, A 0, B 90, C 0} C_DIS
LIN {X 55.62, Y 22.52, Z 90.0, A 0, B 90, C 0} C_DIS
LIN {X 54.43, Y 25.19, Z 90.0, A 0, B 90, C 0} C_DIS
LIN {X 54.06, Y 26.03, Z 90.0, A 0, B 90, C 0} C_DIS
LIN {X 52.71, Y 28.62, Z 90.0, A 0, B 90, C 0} C_DIS
LIN {X 52.28, Y 29.44, Z 90.0, A 0, B 90, C 0} C_DIS
LIN {X 50.76, Y 31.94, Z 90.0, A 0, B 90, C 0} C_DIS
LIN {X 50.29, Y 32.73, Z 90.0, A 0, B 90, C 0} C_DIS
LIN {X 48.61, Y 35.13, Z 90.0, A 0, B 90, C 0} C_DIS
LIN {X 48.08, Y 35.89, Z 90.0, A 0, B 90, C 0} C_DIS
LIN {X 46.26, Y 38.17, Z 90.0, A 0, B 90, C 0} C_DIS
LIN {X 45.69, Y 38.89, Z 90.0, A 0, B 90, C 0} C_DIS
LIN {X 43.72, Y 41.06, Z 90.0, A 0, B 90, C 0} C_DIS
LIN {X 43.1, Y 41.74, Z 90.0, A 0, B 90, C 0} C_DIS
LIN {X 41.0, Y 43.77, Z 90.0, A 0, B 90, C 0} C_DIS
LIN {X 40.34, Y 44.42, Z 90.0, A 0, B 90, C 0} C_DIS
LIN {X 38.11, Y 46.31, Z 90.0, A 0, B 90, C 0} C_DIS
LIN {X 37.41, Y 46.91, Z 90.0, A 0, B 90, C 0} C_DIS
LIN {X 35.07, Y 48.66, Z 90.0, A 0, B 90, C 0} C_DIS
LIN {X 34.33, Y 49.21, Z 90.0, A 0, B 90, C 0} C_DIS
LIN {X 31.88, Y 50.8, Z 90.0, A 0, B 90, C 0} C_DIS
LIN {X 31.1, Y 51.31, Z 90.0, A 0, B 90, C 0} C_DIS
LIN {X 28.56, Y 52.74, Z 90.0, A 0, B 90, C 0} C_DIS
LIN {X 27.75, Y 53.2, Z 90.0, A 0, B 90, C 0} C_DIS
LIN {X 25.12, Y 54.46, Z 90.0, A 0, B 90, C 0} C_DIS
LIN {X 24.29, Y 54.86, Z 90.0, A 0, B 90, C 0} C_DIS
LIN {X 21.58, Y 55.96, Z 90.0, A 0, B 90, C 0} C_DIS
LIN {X 20.72, Y 56.31, Z 90.0, A 0, B 90, C 0} C_DIS
LIN {X 17.95, Y 57.23, Z 90.0, A 0, B 90, C 0} C_DIS
LIN {X 17.07, Y 57.52, Z 90.0, A 0, B 90, C 0} C_DIS
LIN {X 14.24, Y 58.26, Z 90.0, A 0, B 90, C 0} C_DIS
LIN {X 13.35, Y 58.5, Z 90.0, A 0, B 90, C 0} C_DIS
LIN {X 10.48, Y 59.05, Z 90.0, A 0, B 90, C 0} C_DIS
LIN {X 9.58, Y 59.23, Z 90.0, A 0, B 90, C 0} C_DIS
LIN {X 6.68, Y 59.6, Z 90.0, A 0, B 90, C 0} C_DIS
LIN {X 5.76, Y 59.72, Z 90.0, A 0, B 90, C 0} C_DIS
LIN {X 2.84, Y 59.91, Z 90.0, A 0, B 90, C 0} C_DIS
LIN {X 1.92, Y 59.97, Z 90.0, A 0, B 90, C 0} C_DIS
LIN {X -1.0, Y 59.97, Z 90.0, A 0, B 90, C 0} C_DIS
LIN {X -1.92, Y 59.97, Z 90.0, A 0, B 90, C 0} C_DIS
LIN {X -4.84, Y 59.78, Z 90.0, A 0, B 90, C 0} C_DIS
LIN {X -5.76, Y 59.72, Z 90.0, A 0, B 90, C 0} C_DIS
LIN {X -8.66, Y 59.35, Z 90.0, A 0, B 90, C 0} C_DIS
LIN {X -9.58, Y 59.23, Z 90.0, A 0, B 90, C 0} C_DIS
LIN {X -12.45, Y 58.67, Z 90.0, A 0, B 90, C 0} C_DIS
LIN {X -13.35, Y 58.5, Z 90.0, A 0, B 90, C 0} C_DIS
LIN {X -16.18, Y 57.75, Z 90.0, A 0, B 90, C 0} C_DIS
LIN {X -17.07, Y 57.52, Z 90.0, A 0, B 90, C 0} C_DIS
LIN {X -19.85, Y 56.6, Z 90.0, A 0, B 90, C 0} C_DIS
LIN {X -20.72, Y 56.31, Z 90.0, A 0, B 90, C 0} C_DIS
LIN {X -23.43, Y 55.21, Z 90.0, A 0, B 90, C 0} C_DIS
LIN {X -24.29, Y 54.86, Z 90.0, A 0, B 90, C 0} C_DIS
LIN {X -26.92, Y 53.6, Z 90.0, A 0, B 90, C 0} C_DIS
LIN {X -27.75, Y 53.2, Z 90.0, A 0, B 90, C 0} C_DIS
LIN {X -30.3, Y 51.76, Z 90.0, A 0, B 90, C 0} C_DIS
LIN {X -31.1, Y 51.31, Z 90.0, A 0, B 90, C 0} C_DIS
LIN {X -33.55, Y 49.71, Z 90.0, A 0, B 90, C 0} C_DIS
LIN {X -34.33, Y 49.21, Z 90.0, A 0, B 90, C 0} C_DIS
LIN {X -36.67, Y 47.46, Z 90.0, A 0, B 90, C 0} C_DIS
LIN {X -37.41, Y 46.91, Z 90.0, A 0, B 90, C 0} C_DIS
LIN {X -39.64, Y 45.02, Z 90.0, A 0, B 90, C 0} C_DIS
LIN {X -40.34, Y 44.42, Z 90.0, A 0, B 90, C 0} C_DIS
LIN {X -42.44, Y 42.38, Z 90.0, A 0, B 90, C 0} C_DIS
LIN {X -43.1, Y 41.74, Z 90.0, A 0, B 90, C 0} C_DIS
LIN {X -45.07, Y 39.58, Z 90.0, A 0, B 90, C 0} C_DIS
LIN {X -45.69, Y 38.89, Z 90.0, A 0, B 90, C 0} C_DIS
LIN {X -47.51, Y 36.61, Z 90.0, A 0, B 90, C 0} C_DIS
LIN {X -48.08, Y 35.89, Z 90.0, A 0, B 90, C 0} C_DIS
LIN {X -49.76, Y 33.49, Z 90.0, A 0, B 90, C 0} C_DIS
LIN {X -50.29, Y 32.73, Z 90.0, A 0, B 90, C 0} C_DIS
LIN {X -51.8, Y 30.23, Z 90.0, A 0, B 90, C 0} C_DIS
LIN {X -52.28, Y 29.44, Z 90.0, A 0, B 90, C 0} C_DIS
LIN {X -53.63, Y 26.85, Z 90.0, A 0, B 90, C 0} C_DIS
LIN {X -54.06, Y 26.03, Z 90.0, A 0, B 90, C 0} C_DIS
LIN {X -55.24, Y 23.36, Z 90.0, A 0, B 90, C 0} C_DIS
LIN {X -55.62, Y 22.52, Z 90.0, A 0, B 90, C 0} C_DIS
LIN {X -56.62, Y 19.77, Z 90.0, A 0, B 90, C 0} C_DIS
LIN {X -56.94, Y 18.91, Z 90.0, A 0, B 90, C 0} C_DIS
LIN {X -57.78, Y 16.1, Z 90.0, A 0, B 90, C 0} C_DIS
LIN {X -58.04, Y 15.22, Z 90.0, A 0, B 90, C 0} C_DIS
LIN {X -58.69, Y 12.37, Z 90.0, A 0, B 90, C 0} C_DIS
LIN {X -58.89, Y 11.47, Z 90.0, A 0, B 90, C 0} C_DIS
LIN {X -59.36, Y 8.58, Z 90.0, A 0, B 90, C 0} C_DIS
LIN {X -59.51, Y 7.67, Z 90.0, A 0, B 90, C 0} C_DIS
LIN {X -59.79, Y 4.76, Z 90.0, A 0, B 90, C 0} C_DIS
LIN {X -59.88, Y 3.84, Z 90.0, A 0, B 90, C 0} C_DIS
LIN {X -59.97, Y 0.92, Z 90.0, A 0, B 90, C 0} C_DIS
LIN {X -60.0, Y -0.0, Z 90.0, A 0, B 90, C 0} C_DIS
LIN {X -59.91, Y -2.92, Z 90.0, A 0, B 90, C 0} C_DIS
LIN {X -59.88, Y -3.84, Z 90.0, A 0, B 90, C 0} C_DIS
LIN {X -59.6, Y -6.75, Z 90.0, A 0, B 90, C 0} C_DIS
LIN {X -59.51, Y -7.67, Z 90.0, A 0, B 90, C 0} C_DIS
LIN {X -59.04, Y -10.56, Z 90.0, A 0, B 90, C 0} C_DIS
LIN {X -58.89, Y -11.47, Z 90.0, A 0, B 90, C 0} C_DIS
LIN {X -58.24, Y -14.32, Z 90.0, A 0, B 90, C 0} C_DIS
LIN {X -58.04, Y -15.22, Z 90.0, A 0, B 90, C 0} C_DIS
LIN {X -57.21, Y -18.02, Z 90.0, A 0, B 90, C 0} C_DIS
LIN {X -56.94, Y -18.91, Z 90.0, A 0, B 90, C 0} C_DIS
LIN {X -55.93, Y -21.65, Z 90.0, A 0, B 90, C 0} C_DIS
LIN {X -55.62, Y -22.52, Z 90.0, A 0, B 90, C 0} C_DIS
LIN {X -54.43, Y -25.19, Z 90.0, A 0, B 90, C 0} C_DIS
LIN {X -54.06, Y -26.03, Z 90.0, A 0, B 90, C 0} C_DIS
LIN {X -52.71, Y -28.62, Z 90.0, A 0, B 90, C 0} C_DIS
LIN {X -52.28, Y -29.44, Z 90.0, A 0, B 90, C 0} C_DIS
LIN {X -50.76, Y -31.94, Z 90.0, A 0, B 90, C 0} C_DIS
LIN {X -50.29, Y -32.73, Z 90.0, A 0, B 90, C 0} C_DIS
LIN {X -48.61, Y -35.13, Z 90.0, A 0, B 90, C 0} C_DIS
LIN {X -48.08, Y -35.89, Z 90.0, A 0, B 90, C 0} C_DIS
LIN {X -46.26, Y -38.17, Z 90.0, A 0, B 90, C 0} C_DIS
LIN {X -45.69, Y -38.89, Z 90.0, A 0, B 90, C 0} C_DIS
LIN {X -43.72, Y -41.06, Z 90.0, A 0, B 90, C 0} C_DIS
LIN {X -43.1, Y -41.74, Z 90.0, A 0, B 90, C 0} C_DIS
LIN {X -41.0, Y -43.77, Z 90.0, A 0, B 90, C 0} C_DIS
LIN {X -40.34, Y -44.42, Z 90.0, A 0, B 90, C 0} C_DIS
LIN {X -38.11, Y -46.31, Z 90.0, A 0, B 90, C 0} C_DIS
LIN {X -37.41, Y -46.91, Z 90.0, A 0, B 90, C 0} C_DIS
LIN {X -35.07, Y -48.66, Z 90.0, A 0, B 90, C 0} C_DIS
$OUT[1] = FALSE

